LIN {X 0.064,Y -465.840,Z 820.018,A 0.000,B 0.000,C 90.000,E1 219.277} C_DIS
LIN {X -0.205,Y -462.583,Z 820.010,A 0.000,B 0.000,C 90.000,E1 217.729} C_DIS
LIN {X 0.196,Y -459.320,Z 820.001,A 0.000,B 0.000,C 90.000,E1 216.091} C_DIS
LIN {X -0.112,Y -456.022,Z 819.992,A 0.000,B 0.000,C 90.000,E1 214.532} C_DIS
LIN {X 0.155,Y -450.639,Z 819.978,A 0.000,B 0.000,C 90.000,E1 211.926} C_DIS
LIN {X 0.021,Y -446.616,Z 819.967,A 0.000,B 0.000,C 90.000,E1 210.001} C_DIS
LIN {X 0.126,Y -443.411,Z 819.958,A 0.000,B 0.000,C 90.000,E1 208.359} C_DIS
LIN {X -0.002,Y -439.571,Z 819.947,A 0.000,B 0.000,C 90.000,E1 206.411} C_DIS
LIN {X 0.099,Y -437.621,Z 819.941,A 0.000,B 0.000,C 90.000,E1 205.412} C_DIS
LIN {X 0.024,Y -434.306,Z 819.932,A 0.000,B 0.000,C 90.000,E1 203.770} C_DIS
LIN {X 0.087,Y -430.412,Z 819.921,A 0.000,B 0.000,C 90.000,E1 201.770} C_DIS
LIN {X 0.138,Y -426.596,Z 819.910,A 0.000,B 0.000,C 90.000,E1 199.758} C_DIS
LIN {X -0.092,Y -423.266,Z 819.901,A 0.000,B 0.000,C 90.000,E1 198.109} C_DIS
LIN {X -0.075,Y -419.349,Z 819.889,A 0.000,B 0.000,C 90.000,E1 196.079} C_DIS
LIN {X 0.146,Y -415.472,Z 819.878,A 0.000,B 0.000,C 90.000,E1 194.008} C_DIS
LIN {X 0.141,Y -412.294,Z 819.868,A 0.000,B 0.000,C 90.000,E1 192.299} C_DIS
LIN {X 0.007,Y -408.308,Z 819.857,A 0.000,B 0.000,C 90.000,E1 190.254} C_DIS
LIN {X 0.096,Y -405.067,Z 819.847,A 0.000,B 0.000,C 90.000,E1 188.511} C_DIS
LIN {X 0.058,Y -401.826,Z 819.838,A 0.000,B 0.000,C 90.000,E1 186.777} C_DIS
LIN {X 0.025,Y -395.279,Z 819.816,A 0.000,B 0.000,C 90.000,E1 182.922} C_DIS
LIN {X 0.015,Y -392.207,Z 819.805,A 0.000,B 0.000,C 90.000,E1 180.802} C_DIS
LIN {X 0.152,Y -388.677,Z 819.789,A 0.000,B 0.000,C 90.000,E1 177.936} C_DIS
LIN {X 0.084,Y -386.545,Z 819.779,A 0.000,B 0.000,C 90.000,E1 176.159} C_DIS
LIN {X -0.093,Y -384.076,Z 819.767,A 0.000,B 0.000,C 90.000,E1 174.033} C_DIS
LIN {X -0.125,Y -380.731,Z 819.749,A 0.000,B 0.000,C 90.000,E1 170.792} C_DIS
LIN {X 0.144,Y -378.740,Z 819.737,A 0.000,B 0.000,C 90.000,E1 168.578} C_DIS
LIN {X -0.067,Y -376.335,Z 819.721,A 0.000,B 0.000,C 90.000,E1 165.700} C_DIS
LIN {X 0.130,Y -373.483,Z 819.682,A 0.000,B 0.000,C 90.000,E1 158.720} C_DIS
LIN {X -0.016,Y -374.195,Z 819.668,A 0.000,B 0.000,C 90.000,E1 156.177} C_DIS
LIN {X 0.047,Y -376.178,Z 819.656,A 0.000,B 0.000,C 90.000,E1 153.973} C_DIS
LIN {X -0.036,Y -377.112,Z 819.651,A 0.000,B 0.000,C 90.000,E1 153.256} C_DIS
LIN {X 0.026,Y -379.071,Z 819.645,A 0.000,B 0.000,C 90.000,E1 152.153} C_DIS
LIN {X -0.028,Y -380.633,Z 819.641,A 0.000,B 0.000,C 90.000,E1 151.435} C_DIS
LIN {X 0.156,Y -383.722,Z 819.635,A 0.000,B 0.000,C 90.000,E1 150.333} C_DIS
LIN {X 0.046,Y -384.906,Z 819.633,A 0.000,B 0.000,C 90.000,E1 149.999} C_DIS
LIN {X 0.035,Y -387.998,Z 819.629,A 0.000,B 0.000,C 90.000,E1 149.282} C_DIS
LIN {X -0.197,Y -390.381,Z 819.627,A 0.000,B 0.000,C 90.000,E1 148.869} C_DIS
LIN {X 0.187,Y -392.330,Z 819.625,A 0.000,B 0.000,C 90.000,E1 148.456} C_DIS
LIN {X 0.040,Y -394.553,Z 819.623,A 0.000,B 0.000,C 90.000,E1 148.122} C_DIS
LIN {X -0.108,Y -399.019,Z 819.620,A 0.000,B 0.000,C 90.000,E1 147.582} C_DIS
LIN {X -0.132,Y -406.021,Z 819.616,A 0.000,B 0.000,C 90.000,E1 146.834} C_DIS
LIN {X 0.106,Y -413.015,Z 819.612,A 0.000,B 0.000,C 90.000,E1 146.215} C_DIS
LIN {X 0.082,Y -426.154,Z 819.607,A 0.000,B 0.000,C 90.000,E1 145.261} C_DIS
LIN {X -0.035,Y -435.967,Z 819.603,A 0.000,B 0.000,C 90.000,E1 144.609} C_DIS
LIN {X -0.214,Y -446.937,Z 819.599,A 0.000,B 0.000,C 90.000,E1 143.783} C_DIS
LIN {X 0.166,Y -452.778,Z 819.596,A 0.000,B 0.000,C 90.000,E1 143.210} C_DIS
LIN {X -0.262,Y -456.921,Z 819.593,A 0.000,B 0.000,C 90.000,E1 142.844} C_DIS
LIN {X 0.206,Y -462.297,Z 819.590,A 0.000,B 0.000,C 90.000,E1 142.190} C_DIS
LIN {X -0.274,Y -471.185,Z 819.584,A 0.000,B 0.000,C 90.000,E1 141.170} C_DIS
LIN {X 0.222,Y -474.561,Z 819.582,A 0.000,B 0.000,C 90.000,E1 140.642} C_DIS
LIN {X 0.087,Y -477.926,Z 819.579,A 0.000,B 0.000,C 90.000,E1 140.194} C_DIS
LIN {X -0.230,Y -483.509,Z 819.575,A 0.000,B 0.000,C 90.000,E1 139.461} C_DIS
LIN {X -0.288,Y -487.498,Z 819.571,A 0.000,B 0.000,C 90.000,E1 138.852} C_DIS
LIN {X -0.067,Y -490.481,Z 819.569,A 0.000,B 0.000,C 90.000,E1 138.366} C_DIS
LIN {X 0.018,Y -494.875,Z 819.564,A 0.000,B 0.000,C 90.000,E1 137.595} C_DIS
LIN {X 0.001,Y -500.954,Z 819.559,A 0.000,B 0.000,C 90.000,E1 136.539} C_DIS
LIN {X -0.074,Y -505.578,Z 819.554,A 0.000,B 0.000,C 90.000,E1 135.648} C_DIS
LIN {X 0.026,Y -508.795,Z 819.550,A 0.000,B 0.000,C 90.000,E1 135.040} C_DIS
LIN {X -0.194,Y -513.933,Z 819.545,A 0.000,B 0.000,C 90.000,E1 134.028} C_DIS
LIN {X -0.063,Y -520.525,Z 819.537,A 0.000,B 0.000,C 90.000,E1 132.690} C_DIS
LIN {X 0.164,Y -523.164,Z 819.534,A 0.000,B 0.000,C 90.000,E1 132.081} C_DIS
LIN {X 0.094,Y -528.588,Z 819.527,A 0.000,B 0.000,C 90.000,E1 130.782} C_DIS
LIN {X -0.065,Y -532.865,Z 819.520,A 0.000,B 0.000,C 90.000,E1 129.644} C_DIS
LIN {X 0.246,Y -536.671,Z 819.514,A 0.000,B 0.000,C 90.000,E1 128.463} C_DIS
LIN {X -0.158,Y -539.163,Z 819.509,A 0.000,B 0.000,C 90.000,E1 127.649} C_DIS
LIN {X -0.112,Y -541.425,Z 819.504,A 0.000,B 0.000,C 90.000,E1 126.790} C_DIS
LIN {X -0.066,Y -542.850,Z 819.501,A 0.000,B 0.000,C 90.000,E1 126.217} C_DIS
LIN {X -0.011,Y -544.045,Z 819.498,A 0.000,B 0.000,C 90.000,E1 125.644} C_DIS
LIN {X -0.263,Y -544.826,Z 819.495,A 0.000,B 0.000,C 90.000,E1 125.105} C_DIS
LIN {X -0.194,Y -545.485,Z 819.492,A 0.000,B 0.000,C 90.000,E1 124.532} C_DIS
LIN {X 0.133,Y -546.070,Z 819.484,A 0.000,B 0.000,C 90.000,E1 123.086} C_DIS
LIN {X -0.318,Y -547.175,Z 819.478,A 0.000,B 0.000,C 90.000,E1 122.005} C_DIS
LIN {X -0.036,Y -547.993,Z 819.473,A 0.000,B 0.000,C 90.000,E1 121.131} C_DIS
LIN {X -0.253,Y -548.782,Z 819.470,A 0.000,B 0.000,C 90.000,E1 120.590} C_DIS
LIN {X 0.253,Y -549.304,Z 819.468,A 0.000,B 0.000,C 90.000,E1 120.256} C_DIS
LIN {X 0.009,Y -549.680,Z 819.467,A 0.000,B 0.000,C 90.000,E1 120.001} C_DIS
LIN {X -0.078,Y -550.090,Z 819.464,A 0.000,B 0.000,C 90.000,E1 119.589} C_DIS
LIN {X 0.045,Y -550.848,Z 819.462,A 0.000,B 0.000,C 90.000,E1 119.155} C_DIS
LIN {X -0.044,Y -551.594,Z 819.461,A 0.000,B 0.000,C 90.000,E1 119.027} C_DIS
LIN {X -0.011,Y -552.319,Z 819.460,A 0.000,B 0.000,C 90.000,E1 118.743} C_DIS
LIN {X -0.094,Y -552.319,Z 819.458,A 0.000,B 0.000,C 90.000,E1 118.437} C_DIS
LIN {X 0.001,Y -552.285,Z 819.458,A 0.000,B 0.000,C 90.000,E1 118.409} C_DIS
LIN {X -0.042,Y -552.280,Z 819.458,A 0.000,B 0.000,C 90.000,E1 118.409} C_DIS
LIN {X 0.017,Y -552.707,Z 819.457,A 0.000,B 0.000,C 90.000,E1 118.180} C_DIS
LIN {X 0.050,Y -553.492,Z 819.455,A 0.000,B 0.000,C 90.000,E1 117.897} C_DIS
LIN {X -0.064,Y -553.553,Z 819.454,A 0.000,B 0.000,C 90.000,E1 117.769} C_DIS
LIN {X -0.131,Y -554.947,Z 819.450,A 0.000,B 0.000,C 90.000,E1 117.078} C_DIS
LIN {X -0.256,Y -556.790,Z 819.444,A 0.000,B 0.000,C 90.000,E1 115.976} C_DIS
LIN {X 0.136,Y -558.183,Z 819.438,A 0.000,B 0.000,C 90.000,E1 114.823} C_DIS
LIN {X -0.121,Y -559.816,Z 819.430,A 0.000,B 0.000,C 90.000,E1 113.462} C_DIS
LIN {X -0.127,Y -561.223,Z 819.423,A 0.000,B 0.000,C 90.000,E1 112.078} C_DIS
LIN {X -0.124,Y -562.087,Z 819.417,A 0.000,B 0.000,C 90.000,E1 110.972} C_DIS
LIN {X -0.112,Y -562.630,Z 819.410,A 0.000,B 0.000,C 90.000,E1 109.866} C_DIS
LIN {X -0.147,Y -562.902,Z 819.403,A 0.000,B 0.000,C 90.000,E1 108.489} C_DIS
LIN {X 0.070,Y -563.250,Z 819.390,A 0.000,B 0.000,C 90.000,E1 106.260} C_DIS
LIN {X 0.206,Y -564.671,Z 819.372,A 0.000,B 0.000,C 90.000,E1 102.939} C_DIS
LIN {X 0.268,Y -565.893,Z 819.361,A 0.000,B 0.000,C 90.000,E1 101.007} C_DIS
LIN {X 0.159,Y -567.308,Z 819.351,A 0.000,B 0.000,C 90.000,E1 99.095} C_DIS
LIN {X -0.005,Y -568.419,Z 819.342,A 0.000,B 0.000,C 90.000,E1 97.466} C_DIS
LIN {X 0.262,Y -569.428,Z 819.332,A 0.000,B 0.000,C 90.000,E1 95.796} C_DIS
LIN {X -0.063,Y -570.191,Z 819.323,A 0.000,B 0.000,C 90.000,E1 94.188} C_DIS
LIN {X 0.069,Y -570.727,Z 819.316,A 0.000,B 0.000,C 90.000,E1 92.808} C_DIS
LIN {X 0.043,Y -571.139,Z 819.310,A 0.000,B 0.000,C 90.000,E1 91.718} C_DIS
LIN {X 0.141,Y -571.612,Z 819.302,A 0.000,B 0.000,C 90.000,E1 90.344} C_DIS
LIN {X -0.048,Y -572.109,Z 819.291,A 0.000,B 0.000,C 90.000,E1 88.453} C_DIS
LIN {X 0.081,Y -572.499,Z 819.284,A 0.000,B 0.000,C 90.000,E1 87.078} C_DIS
LIN {X -0.009,Y -572.878,Z 819.273,A 0.000,B 0.000,C 90.000,E1 85.179} C_DIS
LIN {X -0.082,Y -573.162,Z 819.263,A 0.000,B 0.000,C 90.000,E1 83.280} C_DIS
LIN {X -0.206,Y -573.573,Z 819.254,A 0.000,B 0.000,C 90.000,E1 81.659} C_DIS
LIN {X 0.242,Y -574.013,Z 819.245,A 0.000,B 0.000,C 90.000,E1 79.982} C_DIS
LIN {X 0.331,Y -574.389,Z 819.235,A 0.000,B 0.000,C 90.000,E1 78.342} C_DIS
LIN {X 0.231,Y -574.657,Z 819.228,A 0.000,B 0.000,C 90.000,E1 76.992} C_DIS
LIN {X -0.229,Y -574.764,Z 819.219,A 0.000,B 0.000,C 90.000,E1 75.408} C_DIS
LIN {X -0.043,Y -574.803,Z 819.211,A 0.000,B 0.000,C 90.000,E1 74.031} C_DIS
LIN {X -0.018,Y -574.673,Z 819.201,A 0.000,B 0.000,C 90.000,E1 72.127} C_DIS
LIN {X -0.198,Y -574.365,Z 819.190,A 0.000,B 0.000,C 90.000,E1 70.242} C_DIS
LIN {X -0.011,Y -573.965,Z 819.181,A 0.000,B 0.000,C 90.000,E1 68.592} C_DIS
LIN {X 0.008,Y -573.527,Z 819.174,A 0.000,B 0.000,C 90.000,E1 67.230} C_DIS
LIN {X 0.013,Y -572.980,Z 819.166,A 0.000,B 0.000,C 90.000,E1 65.869} C_DIS
LIN {X -0.282,Y -572.384,Z 819.158,A 0.000,B 0.000,C 90.000,E1 64.537} C_DIS
LIN {X 0.180,Y -571.631,Z 819.151,A 0.000,B 0.000,C 90.000,E1 63.127} C_DIS
LIN {X 0.288,Y -570.867,Z 819.145,A 0.000,B 0.000,C 90.000,E1 62.025} C_DIS
LIN {X -0.114,Y -569.952,Z 819.139,A 0.000,B 0.000,C 90.000,E1 60.973} C_DIS
LIN {X -0.033,Y -568.780,Z 819.133,A 0.000,B 0.000,C 90.000,E1 59.871} C_DIS
LIN {X -0.178,Y -567.446,Z 819.127,A 0.000,B 0.000,C 90.000,E1 58.791} C_DIS
LIN {X 0.251,Y -565.487,Z 819.119,A 0.000,B 0.000,C 90.000,E1 57.375} C_DIS
LIN {X 0.060,Y -563.654,Z 819.113,A 0.000,B 0.000,C 90.000,E1 56.294} C_DIS
LIN {X 0.153,Y -561.489,Z 819.107,A 0.000,B 0.000,C 90.000,E1 55.182} C_DIS
LIN {X -0.242,Y -559.066,Z 819.101,A 0.000,B 0.000,C 90.000,E1 54.116} C_DIS
LIN {X 0.030,Y -557.004,Z 819.096,A 0.000,B 0.000,C 90.000,E1 53.256} C_DIS
LIN {X -0.061,Y -554.683,Z 819.091,A 0.000,B 0.000,C 90.000,E1 52.431} C_DIS
LIN {X -0.282,Y -552.076,Z 819.087,A 0.000,B 0.000,C 90.000,E1 51.618} C_DIS
LIN {X 0.191,Y -550.176,Z 819.084,A 0.000,B 0.000,C 90.000,E1 51.009} C_DIS
LIN {X -0.069,Y -546.997,Z 819.079,A 0.000,B 0.000,C 90.000,E1 50.194} C_DIS
LIN {X 0.050,Y -543.508,Z 819.074,A 0.000,B 0.000,C 90.000,E1 49.337} C_DIS
LIN {X 0.047,Y -540.939,Z 819.071,A 0.000,B 0.000,C 90.000,E1 48.771} C_DIS
LIN {X -0.328,Y -538.176,Z 819.068,A 0.000,B 0.000,C 90.000,E1 48.243} C_DIS
LIN {X 0.211,Y -534.326,Z 819.064,A 0.000,B 0.000,C 90.000,E1 47.472} C_DIS
LIN {X 0.151,Y -530.947,Z 819.061,A 0.000,B 0.000,C 90.000,E1 46.905} C_DIS
LIN {X -0.294,Y -527.208,Z 819.057,A 0.000,B 0.000,C 90.000,E1 46.377} C_DIS
LIN {X -0.025,Y -523.059,Z 819.054,A 0.000,B 0.000,C 90.000,E1 45.769} C_DIS
LIN {X 0.066,Y -518.885,Z 819.051,A 0.000,B 0.000,C 90.000,E1 45.202} C_DIS
LIN {X 0.048,Y -514.196,Z 819.048,A 0.000,B 0.000,C 90.000,E1 44.636} C_DIS
LIN {X -0.274,Y -507.621,Z 819.044,A 0.000,B 0.000,C 90.000,E1 43.947} C_DIS
LIN {X 0.209,Y -503.531,Z 819.042,A 0.000,B 0.000,C 90.000,E1 43.461} C_DIS
LIN {X 0.086,Y -499.288,Z 819.039,A 0.000,B 0.000,C 90.000,E1 43.056} C_DIS
LIN {X -0.048,Y -492.095,Z 819.036,A 0.000,B 0.000,C 90.000,E1 42.405} C_DIS
LIN {X 0.065,Y -484.633,Z 819.032,A 0.000,B 0.000,C 90.000,E1 41.757} C_DIS
LIN {X 0.006,Y -478.368,Z 819.029,A 0.000,B 0.000,C 90.000,E1 41.272} C_DIS
LIN {X -0.144,Y -470.550,Z 819.026,A 0.000,B 0.000,C 90.000,E1 40.701} C_DIS
LIN {X 0.100,Y -453.134,Z 819.019,A 0.000,B 0.000,C 90.000,E1 39.402} C_DIS
LIN {X -0.118,Y -424.777,Z 819.007,A 0.000,B 0.000,C 90.000,E1 37.317} C_DIS
LIN {X -0.016,Y -409.437,Z 819.000,A 0.000,B 0.000,C 90.000,E1 36.011} C_DIS
LIN {X 0.126,Y -402.370,Z 818.996,A 0.000,B 0.000,C 90.000,E1 35.311} C_DIS
LIN {X -0.153,Y -398.570,Z 818.994,A 0.000,B 0.000,C 90.000,E1 34.898} C_DIS
LIN {X -0.191,Y -398.539,Z 818.994,A 0.000,B 0.000,C 90.000,E1 34.898} C_DIS
LIN {X 0.065,Y -394.044,Z 818.978,A 0.000,B 0.000,C 90.000,E1 32.005} C_DIS
LIN {X 0.063,Y -392.608,Z 818.974,A 0.000,B 0.000,C 90.000,E1 31.209} C_DIS
LIN {X -0.108,Y -393.788,Z 818.958,A 0.000,B 0.000,C 90.000,E1 28.487} C_DIS
LIN {X -0.013,Y -395.477,Z 818.943,A 0.000,B 0.000,C 90.000,E1 25.643} C_DIS
LIN {X 0.126,Y -397.180,Z 818.929,A 0.000,B 0.000,C 90.000,E1 23.153} C_DIS
LIN {X 0.101,Y -399.800,Z 818.911,A 0.000,B 0.000,C 90.000,E1 19.993} C_DIS
LIN {X 0.170,Y -404.433,Z 818.888,A 0.000,B 0.000,C 90.000,E1 15.788} C_DIS
LIN {X -0.101,Y -408.925,Z 818.871,A 0.000,B 0.000,C 90.000,E1 12.703} C_DIS
LIN {X 0.127,Y -412.414,Z 818.859,A 0.000,B 0.000,C 90.000,E1 10.602} C_DIS
LIN {X 0.011,Y -416.583,Z 818.846,A 0.000,B 0.000,C 90.000,E1 8.219} C_DIS
LIN {X -0.172,Y -420.297,Z 818.834,A 0.000,B 0.000,C 90.000,E1 6.201} C_DIS
LIN {X 0.118,Y -424.066,Z 818.823,A 0.000,B 0.000,C 90.000,E1 4.131} C_DIS
LIN {X 0.126,Y -428.656,Z 818.810,A 0.000,B 0.000,C 90.000,E1 1.776} C_DIS
LIN {X -0.098,Y -434.381,Z 818.795,A 0.000,B 0.000,C 90.000,E1 359.141} C_DIS
LIN {X -0.147,Y -440.536,Z 818.781,A 0.000,B 0.000,C 90.000,E1 356.502} C_DIS
LIN {X 0.215,Y -445.329,Z 818.770,A 0.000,B 0.000,C 90.000,E1 354.489} C_DIS
LIN {X -0.205,Y -450.296,Z 818.759,A 0.000,B 0.000,C 90.000,E1 352.591} C_DIS
LIN {X 0.142,Y -453.740,Z 818.752,A 0.000,B 0.000,C 90.000,E1 351.254} C_DIS
LIN {X 0.189,Y -456.426,Z 818.747,A 0.000,B 0.000,C 90.000,E1 350.443} C_DIS
LIN {X -0.041,Y -457.795,Z 818.745,A 0.000,B 0.000,C 90.000,E1 350.151} C_DIS
LIN {X 0.188,Y -459.714,Z 818.744,A 0.000,B 0.000,C 90.000,E1 349.803} C_DIS
LIN {X -0.030,Y -462.146,Z 818.742,A 0.000,B 0.000,C 90.000,E1 349.511} C_DIS
LIN {X 0.047,Y -463.622,Z 818.741,A 0.000,B 0.000,C 90.000,E1 349.342} C_DIS
LIN {X 0.000,Y -468.296,Z 818.739,A 0.000,B 0.000,C 90.000,E1 348.926} C_DIS
LIN {X 0.276,Y -475.809,Z 818.735,A 0.000,B 0.000,C 90.000,E1 348.342} C_DIS
LIN {X 0.107,Y -491.394,Z 818.730,A 0.000,B 0.000,C 90.000,E1 347.353} C_DIS
LIN {X -0.258,Y -499.351,Z 818.727,A 0.000,B 0.000,C 90.000,E1 346.881} C_DIS
LIN {X 0.108,Y -512.060,Z 818.722,A 0.000,B 0.000,C 90.000,E1 345.992} C_DIS
LIN {X -0.288,Y -524.419,Z 818.717,A 0.000,B 0.000,C 90.000,E1 345.172} C_DIS
LIN {X -0.113,Y -535.161,Z 818.713,A 0.000,B 0.000,C 90.000,E1 344.393} C_DIS
LIN {X 0.163,Y -543.988,Z 818.710,A 0.000,B 0.000,C 90.000,E1 343.685} C_DIS
LIN {X -0.186,Y -549.737,Z 818.707,A 0.000,B 0.000,C 90.000,E1 343.251} C_DIS
LIN {X 0.308,Y -556.798,Z 818.704,A 0.000,B 0.000,C 90.000,E1 342.598} C_DIS
LIN {X 0.235,Y -559.566,Z 818.702,A 0.000,B 0.000,C 90.000,E1 342.362} C_DIS
LIN {X -0.109,Y -566.064,Z 818.699,A 0.000,B 0.000,C 90.000,E1 341.764} C_DIS
LIN {X 0.105,Y -571.119,Z 818.696,A 0.000,B 0.000,C 90.000,E1 341.221} C_DIS
LIN {X 0.202,Y -577.132,Z 818.692,A 0.000,B 0.000,C 90.000,E1 340.550} C_DIS
LIN {X -0.245,Y -580.537,Z 818.690,A 0.000,B 0.000,C 90.000,E1 340.188} C_DIS
LIN {X -0.005,Y -584.747,Z 818.687,A 0.000,B 0.000,C 90.000,E1 339.625} C_DIS
LIN {X 0.000,Y -589.612,Z 818.683,A 0.000,B 0.000,C 90.000,E1 338.954} C_DIS
LIN {X 0.101,Y -593.242,Z 818.680,A 0.000,B 0.000,C 90.000,E1 338.411} C_DIS
LIN {X 0.127,Y -598.251,Z 818.676,A 0.000,B 0.000,C 90.000,E1 337.614} C_DIS
LIN {X 0.127,Y -604.634,Z 818.670,A 0.000,B 0.000,C 90.000,E1 336.561} C_DIS
LIN {X -0.115,Y -611.479,Z 818.663,A 0.000,B 0.000,C 90.000,E1 335.409} C_DIS
LIN {X 0.068,Y -616.650,Z 818.658,A 0.000,B 0.000,C 90.000,E1 334.485} C_DIS
LIN {X 0.013,Y -622.075,Z 818.653,A 0.000,B 0.000,C 90.000,E1 333.461} C_DIS
LIN {X 0.025,Y -626.619,Z 818.648,A 0.000,B 0.000,C 90.000,E1 332.564} C_DIS
LIN {X -0.174,Y -630.858,Z 818.643,A 0.000,B 0.000,C 90.000,E1 331.691} C_DIS
LIN {X -0.083,Y -634.400,Z 818.638,A 0.000,B 0.000,C 90.000,E1 330.923} C_DIS
LIN {X -0.108,Y -640.068,Z 818.631,A 0.000,B 0.000,C 90.000,E1 329.665} C_DIS
LIN {X -0.165,Y -643.186,Z 818.627,A 0.000,B 0.000,C 90.000,E1 328.918} C_DIS
LIN {X -0.118,Y -647.110,Z 818.622,A 0.000,B 0.000,C 90.000,E1 327.916} C_DIS
LIN {X -0.102,Y -649.896,Z 818.618,A 0.000,B 0.000,C 90.000,E1 327.168} C_DIS
LIN {X 0.021,Y -653.278,Z 818.612,A 0.000,B 0.000,C 90.000,E1 326.167} C_DIS
LIN {X 0.005,Y -656.498,Z 818.607,A 0.000,B 0.000,C 90.000,E1 325.182} C_DIS
LIN {X -0.412,Y -660.115,Z 818.600,A 0.000,B 0.000,C 90.000,E1 323.989} C_DIS
LIN {X 0.061,Y -662.884,Z 818.594,A 0.000,B 0.000,C 90.000,E1 322.970} C_DIS
LIN {X -0.326,Y -664.721,Z 818.590,A 0.000,B 0.000,C 90.000,E1 322.271} C_DIS
LIN {X 0.210,Y -666.998,Z 818.585,A 0.000,B 0.000,C 90.000,E1 321.251} C_DIS
LIN {X 0.261,Y -669.150,Z 818.579,A 0.000,B 0.000,C 90.000,E1 320.275} C_DIS
LIN {X 0.343,Y -671.150,Z 818.574,A 0.000,B 0.000,C 90.000,E1 319.299} C_DIS
LIN {X 0.015,Y -673.470,Z 818.567,A 0.000,B 0.000,C 90.000,E1 318.119} C_DIS
LIN {X 0.072,Y -674.802,Z 818.563,A 0.000,B 0.000,C 90.000,E1 317.391} C_DIS
LIN {X -0.254,Y -676.645,Z 818.557,A 0.000,B 0.000,C 90.000,E1 316.215} C_DIS
LIN {X -0.154,Y -677.717,Z 818.553,A 0.000,B 0.000,C 90.000,E1 315.486} C_DIS
LIN {X -0.041,Y -678.688,Z 818.549,A 0.000,B 0.000,C 90.000,E1 314.757} C_DIS
LIN {X 0.164,Y -680.193,Z 818.542,A 0.000,B 0.000,C 90.000,E1 313.542} C_DIS
LIN {X -0.036,Y -681.891,Z 818.534,A 0.000,B 0.000,C 90.000,E1 312.123} C_DIS
LIN {X -0.150,Y -683.438,Z 818.526,A 0.000,B 0.000,C 90.000,E1 310.701} C_DIS
LIN {X -0.226,Y -684.931,Z 818.518,A 0.000,B 0.000,C 90.000,E1 309.277} C_DIS
LIN {X 0.254,Y -686.296,Z 818.510,A 0.000,B 0.000,C 90.000,E1 307.810} C_DIS
LIN {X -0.030,Y -687.700,Z 818.501,A 0.000,B 0.000,C 90.000,E1 306.171} C_DIS
LIN {X 0.078,Y -688.817,Z 818.493,A 0.000,B 0.000,C 90.000,E1 304.739} C_DIS
LIN {X 0.371,Y -689.821,Z 818.485,A 0.000,B 0.000,C 90.000,E1 303.293} C_DIS
LIN {X -0.046,Y -691.000,Z 818.476,A 0.000,B 0.000,C 90.000,E1 301.671} C_DIS
LIN {X 0.047,Y -691.765,Z 818.471,A 0.000,B 0.000,C 90.000,E1 300.718} C_DIS
LIN {X -0.091,Y -692.888,Z 818.462,A 0.000,B 0.000,C 90.000,E1 299.077} C_DIS
LIN {X 0.161,Y -693.875,Z 818.454,A 0.000,B 0.000,C 90.000,E1 297.641} C_DIS
LIN {X 0.364,Y -695.143,Z 818.445,A 0.000,B 0.000,C 90.000,E1 295.976} C_DIS
LIN {X 0.042,Y -696.279,Z 818.437,A 0.000,B 0.000,C 90.000,E1 294.591} C_DIS
LIN {X 0.298,Y -696.456,Z 818.435,A 0.000,B 0.000,C 90.000,E1 294.335} C_DIS
LIN {X 0.146,Y -696.298,Z 818.431,A 0.000,B 0.000,C 90.000,E1 293.643} C_DIS
LIN {X -0.262,Y -695.128,Z 818.429,A 0.000,B 0.000,C 90.000,E1 293.206} C_DIS
LIN {X -0.011,Y -694.378,Z 818.428,A 0.000,B 0.000,C 90.000,E1 292.950} C_DIS
LIN {X 0.112,Y -693.656,Z 818.427,A 0.000,B 0.000,C 90.000,E1 292.823} C_DIS
LIN {X -0.033,Y -692.660,Z 818.426,A 0.000,B 0.000,C 90.000,E1 292.717} C_DIS
LIN {X 0.352,Y -689.102,Z 818.424,A 0.000,B 0.000,C 90.000,E1 292.333} C_DIS
LIN {X -0.142,Y -687.796,Z 818.424,A 0.000,B 0.000,C 90.000,E1 292.259} C_DIS
LIN {X -0.211,Y -685.865,Z 818.423,A 0.000,B 0.000,C 90.000,E1 292.153} C_DIS
LIN {X -0.006,Y -681.676,Z 818.422,A 0.000,B 0.000,C 90.000,E1 291.950} C_DIS
LIN {X -0.377,Y -678.102,Z 818.421,A 0.000,B 0.000,C 90.000,E1 291.844} C_DIS
LIN {X -0.218,Y -672.525,Z 818.420,A 0.000,B 0.000,C 90.000,E1 291.663} C_DIS
LIN {X 0.219,Y -663.517,Z 818.419,A 0.000,B 0.000,C 90.000,E1 291.461} C_DIS
LIN {X 0.186,Y -645.614,Z 818.418,A 0.000,B 0.000,C 90.000,E1 291.173} C_DIS
LIN {X 0.227,Y -635.221,Z 818.417,A 0.000,B 0.000,C 90.000,E1 290.972} C_DIS
LIN {X -0.180,Y -625.486,Z 818.415,A 0.000,B 0.000,C 90.000,E1 290.791} C_DIS
LIN {X 0.041,Y -619.557,Z 818.415,A 0.000,B 0.000,C 90.000,E1 290.610} C_DIS
LIN {X 0.065,Y -612.527,Z 818.413,A 0.000,B 0.000,C 90.000,E1 290.355} C_DIS
LIN {X 0.090,Y -609.015,Z 818.412,A 0.000,B 0.000,C 90.000,E1 290.194} C_DIS
LIN {X 0.055,Y -605.447,Z 818.411,A 0.000,B 0.000,C 90.000,E1 289.993} C_DIS
LIN {X 0.000,Y -605.415,Z 818.411,A 0.000,B 0.000,C 90.000,E1 289.993} C_DIS
LIN {X -0.001,Y -604.757,Z 818.411,A 0.000,B 0.000,C 90.000,E1 289.885} C_DIS
LIN {X -0.210,Y -603.719,Z 818.410,A 0.000,B 0.000,C 90.000,E1 289.758} C_DIS
LIN {X -0.115,Y -603.883,Z 818.408,A 0.000,B 0.000,C 90.000,E1 289.504} C_DIS
LIN {X -0.357,Y -604.282,Z 818.408,A 0.000,B 0.000,C 90.000,E1 289.396} C_DIS
LIN {X -0.254,Y -606.323,Z 818.405,A 0.000,B 0.000,C 90.000,E1 288.960} C_DIS
LIN {X 0.009,Y -608.787,Z 818.403,A 0.000,B 0.000,C 90.000,E1 288.544} C_DIS
LIN {X 0.254,Y -612.122,Z 818.400,A 0.000,B 0.000,C 90.000,E1 288.000} C_DIS
LIN {X -0.279,Y -615.641,Z 818.397,A 0.000,B 0.000,C 90.000,E1 287.402} C_DIS
LIN {X -0.224,Y -619.003,Z 818.392,A 0.000,B 0.000,C 90.000,E1 286.622} C_DIS
LIN {X -0.138,Y -621.783,Z 818.388,A 0.000,B 0.000,C 90.000,E1 285.843} C_DIS
LIN {X 0.024,Y -623.265,Z 818.385,A 0.000,B 0.000,C 90.000,E1 285.315} C_DIS
LIN {X 0.151,Y -625.114,Z 818.381,A 0.000,B 0.000,C 90.000,E1 284.537} C_DIS
LIN {X -0.264,Y -625.907,Z 818.378,A 0.000,B 0.000,C 90.000,E1 284.064} C_DIS
LIN {X -0.066,Y -626.486,Z 818.375,A 0.000,B 0.000,C 90.000,E1 283.536} C_DIS
LIN {X -0.063,Y -626.946,Z 818.371,A 0.000,B 0.000,C 90.000,E1 282.771} C_DIS
LIN {X 0.146,Y -626.576,Z 818.368,A 0.000,B 0.000,C 90.000,E1 282.243} C_DIS
LIN {X 0.148,Y -625.448,Z 818.364,A 0.000,B 0.000,C 90.000,E1 281.478} C_DIS
LIN {X -0.269,Y -624.308,Z 818.361,A 0.000,B 0.000,C 90.000,E1 281.007} C_DIS
LIN {X -0.197,Y -622.920,Z 818.358,A 0.000,B 0.000,C 90.000,E1 280.489} C_DIS
LIN {X -0.019,Y -621.143,Z 818.355,A 0.000,B 0.000,C 90.000,E1 279.962} C_DIS
LIN {X -0.024,Y -618.293,Z 818.352,A 0.000,B 0.000,C 90.000,E1 279.321} C_DIS
LIN {X 0.016,Y -615.359,Z 818.349,A 0.000,B 0.000,C 90.000,E1 278.803} C_DIS
LIN {X 0.127,Y -611.931,Z 818.346,A 0.000,B 0.000,C 90.000,E1 278.276} C_DIS
LIN {X -0.216,Y -609.918,Z 818.345,A 0.000,B 0.000,C 90.000,E1 278.049} C_DIS
LIN {X -0.050,Y -606.491,Z 818.342,A 0.000,B 0.000,C 90.000,E1 277.644} C_DIS
LIN {X 0.162,Y -602.542,Z 818.340,A 0.000,B 0.000,C 90.000,E1 277.239} C_DIS
LIN {X 0.050,Y -601.135,Z 818.340,A 0.000,B 0.000,C 90.000,E1 277.125} C_DIS
LIN {X -0.291,Y -594.573,Z 818.337,A 0.000,B 0.000,C 90.000,E1 276.720} C_DIS
LIN {X 0.085,Y -591.033,Z 818.336,A 0.000,B 0.000,C 90.000,E1 276.486} C_DIS
LIN {X -0.151,Y -585.650,Z 818.335,A 0.000,B 0.000,C 90.000,E1 276.258} C_DIS
LIN {X -0.143,Y -580.431,Z 818.333,A 0.000,B 0.000,C 90.000,E1 276.030} C_DIS
LIN {X 0.186,Y -574.584,Z 818.332,A 0.000,B 0.000,C 90.000,E1 275.796} C_DIS
LIN {X -0.149,Y -568.345,Z 818.332,A 0.000,B 0.000,C 90.000,E1 275.682} C_DIS
LIN {X 0.115,Y -566.392,Z 818.331,A 0.000,B 0.000,C 90.000,E1 275.625} C_DIS
LIN {X -0.048,Y -561.313,Z 818.331,A 0.000,B 0.000,C 90.000,E1 275.625} C_DIS
LIN {X -0.080,Y -553.687,Z 818.331,A 0.000,B 0.000,C 90.000,E1 275.625} C_DIS
LIN {X 0.247,Y -551.917,Z 818.331,A 0.000,B 0.000,C 90.000,E1 275.568} C_DIS
LIN {X 0.215,Y -551.792,Z 818.331,A 0.000,B 0.000,C 90.000,E1 275.568} C_DIS
LIN {X 0.063,Y -550.067,Z 818.329,A 0.000,B 0.000,C 90.000,E1 275.277} C_DIS
LIN {X 0.013,Y -550.055,Z 818.329,A 0.000,B 0.000,C 90.000,E1 275.277} C_DIS
LIN {X -0.257,Y -547.943,Z 818.314,A 0.000,B 0.000,C 90.000,E1 272.465} C_DIS
LIN {X 0.083,Y -546.574,Z 818.303,A 0.000,B 0.000,C 90.000,E1 270.458} C_DIS
LIN {X -0.173,Y -545.183,Z 818.292,A 0.000,B 0.000,C 90.000,E1 268.511} C_DIS
LIN {X 0.142,Y -543.651,Z 818.279,A 0.000,B 0.000,C 90.000,E1 266.216} C_DIS
LIN {X -0.197,Y -542.798,Z 818.271,A 0.000,B 0.000,C 90.000,E1 264.837} C_DIS
LIN {X -0.038,Y -542.261,Z 818.267,A 0.000,B 0.000,C 90.000,E1 263.970} C_DIS
LIN {X 0.200,Y -540.797,Z 818.257,A 0.000,B 0.000,C 90.000,E1 262.243} C_DIS
LIN {X 0.017,Y -539.306,Z 818.248,A 0.000,B 0.000,C 90.000,E1 260.557} C_DIS
LIN {X 0.268,Y -537.902,Z 818.240,A 0.000,B 0.000,C 90.000,E1 259.106} C_DIS
LIN {X 0.122,Y -536.177,Z 818.230,A 0.000,B 0.000,C 90.000,E1 257.409} C_DIS
LIN {X 0.005,Y -534.713,Z 818.222,A 0.000,B 0.000,C 90.000,E1 255.992} C_DIS
LIN {X -0.138,Y -533.063,Z 818.214,A 0.000,B 0.000,C 90.000,E1 254.574} C_DIS
LIN {X 0.014,Y -531.097,Z 818.205,A 0.000,B 0.000,C 90.000,E1 252.834} C_DIS
LIN {X -0.060,Y -529.319,Z 818.197,A 0.000,B 0.000,C 90.000,E1 251.402} C_DIS
LIN {X -0.010,Y -527.896,Z 818.190,A 0.000,B 0.000,C 90.000,E1 250.242} C_DIS
LIN {X 0.196,Y -525.902,Z 818.182,A 0.000,B 0.000,C 90.000,E1 248.773} C_DIS
LIN {X 0.037,Y -523.373,Z 818.173,A 0.000,B 0.000,C 90.000,E1 247.050} C_DIS
LIN {X 0.016,Y -520.710,Z 818.163,A 0.000,B 0.000,C 90.000,E1 245.305} C_DIS
LIN {X -0.128,Y -518.814,Z 818.156,A 0.000,B 0.000,C 90.000,E1 244.152} C_DIS
LIN {X 0.068,Y -516.361,Z 818.148,A 0.000,B 0.000,C 90.000,E1 242.666} C_DIS
LIN {X -0.149,Y -515.391,Z 818.145,A 0.000,B 0.000,C 90.000,E1 242.103} C_DIS
LIN {X -0.127,Y -512.052,Z 818.135,A 0.000,B 0.000,C 90.000,E1 240.333} C_DIS
LIN {X -0.256,Y -509.343,Z 818.127,A 0.000,B 0.000,C 90.000,E1 238.869} C_DIS
LIN {X -0.064,Y -506.958,Z 818.120,A 0.000,B 0.000,C 90.000,E1 237.661} C_DIS
LIN {X 0.048,Y -505.134,Z 818.115,A 0.000,B 0.000,C 90.000,E1 236.755} C_DIS
LIN {X 0.049,Y -501.867,Z 818.107,A 0.000,B 0.000,C 90.000,E1 235.261} C_DIS
LIN {X -0.019,Y -499.109,Z 818.100,A 0.000,B 0.000,C 90.000,E1 234.069} C_DIS
LIN {X 0.297,Y -496.980,Z 818.095,A 0.000,B 0.000,C 90.000,E1 233.130} C_DIS
LIN {X -0.079,Y -493.298,Z 818.087,A 0.000,B 0.000,C 90.000,E1 231.662} C_DIS
LIN {X -0.017,Y -486.156,Z 818.070,A 0.000,B 0.000,C 90.000,E1 228.609} C_DIS
LIN {X -0.018,Y -481.253,Z 818.058,A 0.000,B 0.000,C 90.000,E1 226.458} C_DIS
LIN {X 0.029,Y -479.169,Z 818.053,A 0.000,B 0.000,C 90.000,E1 225.526} C_DIS
LIN {X 0.273,Y -475.783,Z 818.044,A 0.000,B 0.000,C 90.000,E1 223.947} C_DIS
LIN {X -0.212,Y -472.486,Z 818.036,A 0.000,B 0.000,C 90.000,E1 222.447} C_DIS
LIN {X -0.213,Y -467.882,Z 818.024,A 0.000,B 0.000,C 90.000,E1 220.253} C_DIS
LIN {X 0.018,Y -463.271,Z 818.011,A 0.000,B 0.000,C 90.000,E1 218.016} C_DIS
LIN {X 0.173,Y -459.362,Z 818.001,A 0.000,B 0.000,C 90.000,E1 216.091} C_DIS
LIN {X 0.028,Y -457.272,Z 817.995,A 0.000,B 0.000,C 90.000,E1 215.152} C_DIS
LIN {X -0.134,Y -456.062,Z 817.992,A 0.000,B 0.000,C 90.000,E1 214.532} C_DIS
LIN {X 0.045,Y -451.357,Z 817.979,A 0.000,B 0.000,C 90.000,E1 212.260} C_DIS
LIN {X -0.073,Y -447.326,Z 817.969,A 0.000,B 0.000,C 90.000,E1 210.335} C_DIS
LIN {X 0.050,Y -444.088,Z 817.959,A 0.000,B 0.000,C 90.000,E1 208.693} C_DIS
LIN {X -0.100,Y -440.908,Z 817.950,A 0.000,B 0.000,C 90.000,E1 207.078} C_DIS
LIN {X 0.245,Y -438.355,Z 817.943,A 0.000,B 0.000,C 90.000,E1 205.720} C_DIS
LIN {X 0.179,Y -435.064,Z 817.934,A 0.000,B 0.000,C 90.000,E1 204.079} C_DIS
LIN {X 0.096,Y -431.142,Z 817.923,A 0.000,B 0.000,C 90.000,E1 202.099} C_DIS
LIN {X -0.077,Y -427.317,Z 817.912,A 0.000,B 0.000,C 90.000,E1 200.120} C_DIS
LIN {X -0.081,Y -424.709,Z 817.904,A 0.000,B 0.000,C 90.000,E1 198.779} C_DIS
LIN {X 0.150,Y -420.119,Z 817.891,A 0.000,B 0.000,C 90.000,E1 196.386} C_DIS
LIN {X 0.095,Y -416.186,Z 817.880,A 0.000,B 0.000,C 90.000,E1 194.356} C_DIS
LIN {X 0.139,Y -412.398,Z 817.868,A 0.000,B 0.000,C 90.000,E1 192.299} C_DIS
LIN {X 0.007,Y -408.431,Z 817.857,A 0.000,B 0.000,C 90.000,E1 190.254} C_DIS
LIN {X 0.098,Y -405.198,Z 817.847,A 0.000,B 0.000,C 90.000,E1 188.511} C_DIS
LIN {X 0.063,Y -401.933,Z 817.838,A 0.000,B 0.000,C 90.000,E1 186.777} C_DIS
LIN {X 0.201,Y -397.043,Z 817.822,A 0.000,B 0.000,C 90.000,E1 183.955} C_DIS
LIN {X 0.102,Y -392.890,Z 817.807,A 0.000,B 0.000,C 90.000,E1 181.146} C_DIS
LIN {X 0.172,Y -388.846,Z 817.789,A 0.000,B 0.000,C 90.000,E1 177.936} C_DIS
LIN {X -0.179,Y -387.203,Z 817.781,A 0.000,B 0.000,C 90.000,E1 176.560} C_DIS
LIN {X -0.065,Y -384.310,Z 817.767,A 0.000,B 0.000,C 90.000,E1 174.033} C_DIS
LIN {X -0.174,Y -380.664,Z 817.747,A 0.000,B 0.000,C 90.000,E1 170.443} C_DIS
LIN {X 0.091,Y -378.675,Z 817.735,A 0.000,B 0.000,C 90.000,E1 168.229} C_DIS
LIN {X -0.032,Y -376.346,Z 817.719,A 0.000,B 0.000,C 90.000,E1 165.338} C_DIS
LIN {X -0.174,Y -373.755,Z 817.680,A 0.000,B 0.000,C 90.000,E1 158.411} C_DIS
LIN {X 0.065,Y -374.311,Z 817.668,A 0.000,B 0.000,C 90.000,E1 156.177} C_DIS
LIN {X 0.005,Y -375.642,Z 817.658,A 0.000,B 0.000,C 90.000,E1 154.357} C_DIS
LIN {X 0.044,Y -376.884,Z 817.651,A 0.000,B 0.000,C 90.000,E1 153.256} C_DIS
LIN {X 0.104,Y -378.622,Z 817.645,A 0.000,B 0.000,C 90.000,E1 152.153} C_DIS
LIN {X 0.045,Y -380.053,Z 817.641,A 0.000,B 0.000,C 90.000,E1 151.435} C_DIS
LIN {X -0.001,Y -381.866,Z 817.637,A 0.000,B 0.000,C 90.000,E1 150.717} C_DIS
LIN {X 0.018,Y -385.666,Z 817.630,A 0.000,B 0.000,C 90.000,E1 149.459} C_DIS
LIN {X 0.029,Y -387.932,Z 817.627,A 0.000,B 0.000,C 90.000,E1 148.918} C_DIS
LIN {X 0.073,Y -390.421,Z 817.625,A 0.000,B 0.000,C 90.000,E1 148.408} C_DIS
LIN {X -0.123,Y -394.235,Z 817.621,A 0.000,B 0.000,C 90.000,E1 147.788} C_DIS
LIN {X -0.061,Y -397.744,Z 817.618,A 0.000,B 0.000,C 90.000,E1 147.248} C_DIS
LIN {X 0.041,Y -408.167,Z 817.612,A 0.000,B 0.000,C 90.000,E1 146.087} C_DIS
LIN {X -0.115,Y -411.450,Z 817.610,A 0.000,B 0.000,C 90.000,E1 145.801} C_DIS
LIN {X -0.157,Y -422.816,Z 817.605,A 0.000,B 0.000,C 90.000,E1 144.895} C_DIS
LIN {X 0.006,Y -430.662,Z 817.602,A 0.000,B 0.000,C 90.000,E1 144.322} C_DIS
LIN {X -0.234,Y -435.504,Z 817.600,A 0.000,B 0.000,C 90.000,E1 143.989} C_DIS
LIN {X 0.101,Y -442.988,Z 817.596,A 0.000,B 0.000,C 90.000,E1 143.336} C_DIS
LIN {X -0.191,Y -448.740,Z 817.594,A 0.000,B 0.000,C 90.000,E1 142.844} C_DIS
LIN {X 0.011,Y -453.009,Z 817.591,A 0.000,B 0.000,C 90.000,E1 142.396} C_DIS
LIN {X -0.117,Y -458.403,Z 817.588,A 0.000,B 0.000,C 90.000,E1 141.823} C_DIS
LIN {X 0.090,Y -462.225,Z 817.585,A 0.000,B 0.000,C 90.000,E1 141.331} C_DIS
LIN {X 0.122,Y -464.723,Z 817.583,A 0.000,B 0.000,C 90.000,E1 141.009} C_DIS
LIN {X -0.020,Y -468.570,Z 817.581,A 0.000,B 0.000,C 90.000,E1 140.561} C_DIS
LIN {X 0.104,Y -471.048,Z 817.579,A 0.000,B 0.000,C 90.000,E1 140.231} C_DIS
LIN {X 0.098,Y -478.907,Z 817.573,A 0.000,B 0.000,C 90.000,E1 139.138} C_DIS
LIN {X 0.011,Y -483.036,Z 817.570,A 0.000,B 0.000,C 90.000,E1 138.528} C_DIS
LIN {X -0.232,Y -488.637,Z 817.565,A 0.000,B 0.000,C 90.000,E1 137.634} C_DIS
LIN {X -0.001,Y -491.268,Z 817.562,A 0.000,B 0.000,C 90.000,E1 137.148} C_DIS
LIN {X -0.243,Y -498.686,Z 817.554,A 0.000,B 0.000,C 90.000,E1 135.810} C_DIS
LIN {X -0.235,Y -504.238,Z 817.549,A 0.000,B 0.000,C 90.000,E1 134.757} C_DIS
LIN {X 0.329,Y -508.015,Z 817.544,A 0.000,B 0.000,C 90.000,E1 133.947} C_DIS
LIN {X 0.109,Y -513.187,Z 817.539,A 0.000,B 0.000,C 90.000,E1 132.933} C_DIS
LIN {X -0.101,Y -516.048,Z 817.535,A 0.000,B 0.000,C 90.000,E1 132.366} C_DIS
LIN {X 0.089,Y -518.567,Z 817.532,A 0.000,B 0.000,C 90.000,E1 131.757} C_DIS
LIN {X -0.152,Y -522.065,Z 817.527,A 0.000,B 0.000,C 90.000,E1 130.906} C_DIS
LIN {X 0.080,Y -524.242,Z 817.524,A 0.000,B 0.000,C 90.000,E1 130.297} C_DIS
LIN {X 0.232,Y -529.358,Z 817.516,A 0.000,B 0.000,C 90.000,E1 128.830} C_DIS
LIN {X -0.260,Y -532.685,Z 817.510,A 0.000,B 0.000,C 90.000,E1 127.729} C_DIS
LIN {X -0.285,Y -535.830,Z 817.503,A 0.000,B 0.000,C 90.000,E1 126.583} C_DIS
LIN {X 0.162,Y -537.959,Z 817.498,A 0.000,B 0.000,C 90.000,E1 125.678} C_DIS
LIN {X 0.196,Y -539.304,Z 817.494,A 0.000,B 0.000,C 90.000,E1 124.818} C_DIS
LIN {X -0.081,Y -539.984,Z 817.490,A 0.000,B 0.000,C 90.000,E1 124.278} C_DIS
LIN {X -0.034,Y -540.545,Z 817.486,A 0.000,B 0.000,C 90.000,E1 123.420} C_DIS
LIN {X -0.056,Y -542.489,Z 817.479,A 0.000,B 0.000,C 90.000,E1 122.291} C_DIS
LIN {X -0.038,Y -543.136,Z 817.478,A 0.000,B 0.000,C 90.000,E1 122.005} C_DIS
LIN {X 0.096,Y -543.775,Z 817.477,A 0.000,B 0.000,C 90.000,E1 121.799} C_DIS
LIN {X -0.169,Y -544.502,Z 817.475,A 0.000,B 0.000,C 90.000,E1 121.544} C_DIS
LIN {X -0.149,Y -545.072,Z 817.474,A 0.000,B 0.000,C 90.000,E1 121.258} C_DIS
LIN {X -0.326,Y -545.853,Z 817.472,A 0.000,B 0.000,C 90.000,E1 121.003} C_DIS
LIN {X -0.086,Y -547.149,Z 817.469,A 0.000,B 0.000,C 90.000,E1 120.413} C_DIS
LIN {X 0.003,Y -547.928,Z 817.467,A 0.000,B 0.000,C 90.000,E1 120.129} C_DIS
LIN {X 0.260,Y -549.033,Z 817.464,A 0.000,B 0.000,C 90.000,E1 119.539} C_DIS
LIN {X 0.045,Y -550.400,Z 817.461,A 0.000,B 0.000,C 90.000,E1 118.999} C_DIS
LIN {X 0.056,Y -551.601,Z 817.458,A 0.000,B 0.000,C 90.000,E1 118.437} C_DIS
LIN {X -0.110,Y -554.020,Z 817.452,A 0.000,B 0.000,C 90.000,E1 117.334} C_DIS
LIN {X -0.247,Y -556.025,Z 817.446,A 0.000,B 0.000,C 90.000,E1 116.232} C_DIS
LIN {X 0.350,Y -557.256,Z 817.441,A 0.000,B 0.000,C 90.000,E1 115.335} C_DIS
LIN {X 0.305,Y -559.026,Z 817.433,A 0.000,B 0.000,C 90.000,E1 113.951} C_DIS
LIN {X 0.070,Y -560.643,Z 817.426,A 0.000,B 0.000,C 90.000,E1 112.589} C_DIS
LIN {X -0.135,Y -561.939,Z 817.418,A 0.000,B 0.000,C 90.000,E1 111.227} C_DIS
LIN {X -0.118,Y -562.545,Z 817.412,A 0.000,B 0.000,C 90.000,E1 110.120} C_DIS
LIN {X 0.114,Y -562.794,Z 817.407,A 0.000,B 0.000,C 90.000,E1 109.268} C_DIS
LIN {X -0.049,Y -563.048,Z 817.401,A 0.000,B 0.000,C 90.000,E1 108.181} C_DIS
LIN {X -0.144,Y -563.427,Z 817.390,A 0.000,B 0.000,C 90.000,E1 106.260} C_DIS
LIN {X -0.163,Y -564.747,Z 817.373,A 0.000,B 0.000,C 90.000,E1 103.231} C_DIS
LIN {X 0.065,Y -566.153,Z 817.361,A 0.000,B 0.000,C 90.000,E1 101.007} C_DIS
LIN {X -0.037,Y -567.555,Z 817.351,A 0.000,B 0.000,C 90.000,E1 99.095} C_DIS
LIN {X 0.195,Y -568.503,Z 817.343,A 0.000,B 0.000,C 90.000,E1 97.701} C_DIS
LIN {X -0.096,Y -569.500,Z 817.334,A 0.000,B 0.000,C 90.000,E1 96.087} C_DIS
LIN {X -0.206,Y -569.944,Z 817.329,A 0.000,B 0.000,C 90.000,E1 95.277} C_DIS
LIN {X -0.079,Y -570.585,Z 817.322,A 0.000,B 0.000,C 90.000,E1 93.898} C_DIS
LIN {X 0.155,Y -571.213,Z 817.313,A 0.000,B 0.000,C 90.000,E1 92.236} C_DIS
LIN {X 0.273,Y -571.707,Z 817.305,A 0.000,B 0.000,C 90.000,E1 90.859} C_DIS
LIN {X -0.186,Y -572.104,Z 817.297,A 0.000,B 0.000,C 90.000,E1 89.542} C_DIS
LIN {X 0.085,Y -572.553,Z 817.288,A 0.000,B 0.000,C 90.000,E1 87.879} C_DIS
LIN {X 0.093,Y -572.817,Z 817.282,A 0.000,B 0.000,C 90.000,E1 86.788} C_DIS
LIN {X -0.026,Y -573.212,Z 817.272,A 0.000,B 0.000,C 90.000,E1 84.894} C_DIS
LIN {X -0.223,Y -573.468,Z 817.263,A 0.000,B 0.000,C 90.000,E1 83.280} C_DIS
LIN {X 0.030,Y -573.792,Z 817.255,A 0.000,B 0.000,C 90.000,E1 81.894} C_DIS
LIN {X 0.113,Y -574.299,Z 817.244,A 0.000,B 0.000,C 90.000,E1 79.982} C_DIS
LIN {X 0.208,Y -574.667,Z 817.235,A 0.000,B 0.000,C 90.000,E1 78.342} C_DIS
LIN {X 0.113,Y -574.909,Z 817.228,A 0.000,B 0.000,C 90.000,E1 76.992} C_DIS
LIN {X 0.213,Y -574.998,Z 817.219,A 0.000,B 0.000,C 90.000,E1 75.353} C_DIS
LIN {X 0.044,Y -574.974,Z 817.210,A 0.000,B 0.000,C 90.000,E1 73.740} C_DIS
LIN {X 0.238,Y -574.853,Z 817.202,A 0.000,B 0.000,C 90.000,E1 72.362} C_DIS
LIN {X 0.243,Y -574.616,Z 817.193,A 0.000,B 0.000,C 90.000,E1 70.732} C_DIS
LIN {X 0.068,Y -574.294,Z 817.186,A 0.000,B 0.000,C 90.000,E1 69.390} C_DIS
LIN {X 0.259,Y -573.997,Z 817.180,A 0.000,B 0.000,C 90.000,E1 68.284} C_DIS
LIN {X -0.087,Y -573.637,Z 817.174,A 0.000,B 0.000,C 90.000,E1 67.230} C_DIS
LIN {X -0.079,Y -573.060,Z 817.166,A 0.000,B 0.000,C 90.000,E1 65.869} C_DIS
LIN {X 0.143,Y -572.451,Z 817.158,A 0.000,B 0.000,C 90.000,E1 64.485} C_DIS
LIN {X 0.090,Y -571.684,Z 817.151,A 0.000,B 0.000,C 90.000,E1 63.127} C_DIS
LIN {X 0.198,Y -570.875,Z 817.145,A 0.000,B 0.000,C 90.000,E1 62.025} C_DIS
LIN {X 0.295,Y -569.908,Z 817.139,A 0.000,B 0.000,C 90.000,E1 60.923} C_DIS
LIN {X -0.124,Y -568.721,Z 817.133,A 0.000,B 0.000,C 90.000,E1 59.871} C_DIS
LIN {X 0.217,Y -567.347,Z 817.127,A 0.000,B 0.000,C 90.000,E1 58.742} C_DIS
LIN {X 0.159,Y -565.352,Z 817.119,A 0.000,B 0.000,C 90.000,E1 57.375} C_DIS
LIN {X -0.033,Y -563.469,Z 817.113,A 0.000,B 0.000,C 90.000,E1 56.294} C_DIS
LIN {X 0.057,Y -561.238,Z 817.107,A 0.000,B 0.000,C 90.000,E1 55.182} C_DIS
LIN {X 0.112,Y -558.803,Z 817.101,A 0.000,B 0.000,C 90.000,E1 54.069} C_DIS
LIN {X -0.072,Y -556.672,Z 817.096,A 0.000,B 0.000,C 90.000,E1 53.256} C_DIS
LIN {X 0.172,Y -554.297,Z 817.091,A 0.000,B 0.000,C 90.000,E1 52.396} C_DIS
LIN {X -0.047,Y -551.637,Z 817.087,A 0.000,B 0.000,C 90.000,E1 51.582} C_DIS
LIN {X 0.136,Y -548.619,Z 817.082,A 0.000,B 0.000,C 90.000,E1 50.723} C_DIS
LIN {X -0.185,Y -546.458,Z 817.079,A 0.000,B 0.000,C 90.000,E1 50.194} C_DIS
LIN {X 0.090,Y -543.522,Z 817.075,A 0.000,B 0.000,C 90.000,E1 49.461} C_DIS
LIN {X -0.267,Y -540.996,Z 817.072,A 0.000,B 0.000,C 90.000,E1 48.933} C_DIS
LIN {X -0.277,Y -536.636,Z 817.067,A 0.000,B 0.000,C 90.000,E1 48.081} C_DIS
LIN {X -0.100,Y -534.346,Z 817.065,A 0.000,B 0.000,C 90.000,E1 47.634} C_DIS
LIN {X 0.010,Y -530.018,Z 817.061,A 0.000,B 0.000,C 90.000,E1 46.905} C_DIS
LIN {X 0.303,Y -526.186,Z 817.057,A 0.000,B 0.000,C 90.000,E1 46.296} C_DIS
LIN {X 0.188,Y -521.945,Z 817.054,A 0.000,B 0.000,C 90.000,E1 45.729} C_DIS
LIN {X -0.100,Y -518.642,Z 817.052,A 0.000,B 0.000,C 90.000,E1 45.324} C_DIS
LIN {X -0.265,Y -513.791,Z 817.049,A 0.000,B 0.000,C 90.000,E1 44.757} C_DIS
LIN {X 0.159,Y -509.865,Z 817.046,A 0.000,B 0.000,C 90.000,E1 44.271} C_DIS
LIN {X 0.121,Y -504.469,Z 817.043,A 0.000,B 0.000,C 90.000,E1 43.704} C_DIS
LIN {X -0.112,Y -498.825,Z 817.040,A 0.000,B 0.000,C 90.000,E1 43.176} C_DIS
LIN {X 0.129,Y -493.028,Z 817.037,A 0.000,B 0.000,C 90.000,E1 42.609} C_DIS
LIN {X 0.204,Y -486.940,Z 817.034,A 0.000,B 0.000,C 90.000,E1 42.081} C_DIS
LIN {X 0.101,Y -480.751,Z 817.031,A 0.000,B 0.000,C 90.000,E1 41.595} C_DIS
LIN {X 0.027,Y -471.509,Z 817.027,A 0.000,B 0.000,C 90.000,E1 40.906} C_DIS
LIN {X -0.039,Y -463.519,Z 817.024,A 0.000,B 0.000,C 90.000,E1 40.334} C_DIS
LIN {X 0.136,Y -449.239,Z 817.018,A 0.000,B 0.000,C 90.000,E1 39.277} C_DIS
LIN {X 0.018,Y -420.977,Z 817.006,A 0.000,B 0.000,C 90.000,E1 37.156} C_DIS
LIN {X -0.108,Y -408.787,Z 817.001,A 0.000,B 0.000,C 90.000,E1 36.137} C_DIS
LIN {X -0.209,Y -403.015,Z 816.998,A 0.000,B 0.000,C 90.000,E1 35.598} C_DIS
LIN {X 0.202,Y -400.491,Z 816.996,A 0.000,B 0.000,C 90.000,E1 35.231} C_DIS
LIN {X 0.177,Y -398.892,Z 816.995,A 0.000,B 0.000,C 90.000,E1 35.025} C_DIS
LIN {X 0.139,Y -398.849,Z 816.995,A 0.000,B 0.000,C 90.000,E1 35.025} C_DIS
LIN {X 0.033,Y -393.929,Z 816.977,A 0.000,B 0.000,C 90.000,E1 31.926} C_DIS
LIN {X -0.172,Y -392.811,Z 816.974,A 0.000,B 0.000,C 90.000,E1 31.337} C_DIS
LIN {X -0.005,Y -393.891,Z 816.960,A 0.000,B 0.000,C 90.000,E1 28.743} C_DIS
LIN {X -0.080,Y -395.518,Z 816.944,A 0.000,B 0.000,C 90.000,E1 25.924} C_DIS
LIN {X 0.088,Y -397.461,Z 816.928,A 0.000,B 0.000,C 90.000,E1 23.078} C_DIS
LIN {X -0.156,Y -399.745,Z 816.913,A 0.000,B 0.000,C 90.000,E1 20.301} C_DIS
LIN {X -0.069,Y -403.882,Z 816.891,A 0.000,B 0.000,C 90.000,E1 16.441} C_DIS
LIN {X 0.144,Y -408.755,Z 816.872,A 0.000,B 0.000,C 90.000,E1 12.939} C_DIS
LIN {X -0.034,Y -412.201,Z 816.861,A 0.000,B 0.000,C 90.000,E1 10.894} C_DIS
LIN {X -0.154,Y -416.361,Z 816.847,A 0.000,B 0.000,C 90.000,E1 8.511} C_DIS
LIN {X 0.124,Y -420.081,Z 816.836,A 0.000,B 0.000,C 90.000,E1 6.429} C_DIS
LIN {X -0.052,Y -423.194,Z 816.826,A 0.000,B 0.000,C 90.000,E1 4.759} C_DIS
LIN {X -0.096,Y -427.720,Z 816.813,A 0.000,B 0.000,C 90.000,E1 2.407} C_DIS
LIN {X 0.164,Y -433.160,Z 816.799,A 0.000,B 0.000,C 90.000,E1 359.771} C_DIS
LIN {X -0.141,Y -437.580,Z 816.788,A 0.000,B 0.000,C 90.000,E1 357.822} C_DIS
LIN {X -0.026,Y -441.520,Z 816.779,A 0.000,B 0.000,C 90.000,E1 356.159} C_DIS
LIN {X -0.091,Y -446.336,Z 816.768,A 0.000,B 0.000,C 90.000,E1 354.204} C_DIS
LIN {X -0.186,Y -450.488,Z 816.759,A 0.000,B 0.000,C 90.000,E1 352.591} C_DIS
LIN {X -0.146,Y -454.784,Z 816.750,A 0.000,B 0.000,C 90.000,E1 350.971} C_DIS
LIN {X 0.066,Y -455.791,Z 816.748,A 0.000,B 0.000,C 90.000,E1 350.622} C_DIS
LIN {X -0.018,Y -457.593,Z 816.745,A 0.000,B 0.000,C 90.000,E1 350.151} C_DIS
LIN {X -0.001,Y -459.483,Z 816.743,A 0.000,B 0.000,C 90.000,E1 349.803} C_DIS
LIN {X 0.074,Y -460.430,Z 816.742,A 0.000,B 0.000,C 90.000,E1 349.634} C_DIS
LIN {X 0.000,Y -463.174,Z 816.741,A 0.000,B 0.000,C 90.000,E1 349.285} C_DIS
LIN {X -0.113,Y -469.612,Z 816.737,A 0.000,B 0.000,C 90.000,E1 348.701} C_DIS
LIN {X -0.015,Y -473.447,Z 816.736,A 0.000,B 0.000,C 90.000,E1 348.409} C_DIS
LIN {X 0.018,Y -476.533,Z 816.734,A 0.000,B 0.000,C 90.000,E1 348.173} C_DIS
LIN {X -0.170,Y -489.406,Z 816.730,A 0.000,B 0.000,C 90.000,E1 347.353} C_DIS
LIN {X 0.157,Y -498.802,Z 816.726,A 0.000,B 0.000,C 90.000,E1 346.700} C_DIS
LIN {X -0.066,Y -511.520,Z 816.722,A 0.000,B 0.000,C 90.000,E1 345.880} C_DIS
LIN {X 0.198,Y -523.955,Z 816.717,A 0.000,B 0.000,C 90.000,E1 344.991} C_DIS
LIN {X -0.130,Y -534.696,Z 816.713,A 0.000,B 0.000,C 90.000,E1 344.267} C_DIS
LIN {X 0.147,Y -543.551,Z 816.709,A 0.000,B 0.000,C 90.000,E1 343.559} C_DIS
LIN {X -0.249,Y -553.641,Z 816.704,A 0.000,B 0.000,C 90.000,E1 342.779} C_DIS
LIN {X 0.322,Y -559.192,Z 816.702,A 0.000,B 0.000,C 90.000,E1 342.236} C_DIS
LIN {X 0.064,Y -565.738,Z 816.698,A 0.000,B 0.000,C 90.000,E1 341.638} C_DIS
LIN {X 0.273,Y -570.824,Z 816.695,A 0.000,B 0.000,C 90.000,E1 341.094} C_DIS
LIN {X 0.276,Y -576.970,Z 816.691,A 0.000,B 0.000,C 90.000,E1 340.423} C_DIS
LIN {X 0.215,Y -582.495,Z 816.688,A 0.000,B 0.000,C 90.000,E1 339.752} C_DIS
LIN {X 0.270,Y -586.533,Z 816.685,A 0.000,B 0.000,C 90.000,E1 339.209} C_DIS
LIN {X 0.230,Y -592.169,Z 816.680,A 0.000,B 0.000,C 90.000,E1 338.411} C_DIS
LIN {X -0.257,Y -596.442,Z 816.677,A 0.000,B 0.000,C 90.000,E1 337.794} C_DIS
LIN {X -0.281,Y -602.930,Z 816.671,A 0.000,B 0.000,C 90.000,E1 336.741} C_DIS
LIN {X 0.051,Y -608.325,Z 816.666,A 0.000,B 0.000,C 90.000,E1 335.793} C_DIS
LIN {X -0.387,Y -615.065,Z 816.659,A 0.000,B 0.000,C 90.000,E1 334.665} C_DIS
LIN {X 0.104,Y -619.273,Z 816.655,A 0.000,B 0.000,C 90.000,E1 333.845} C_DIS
LIN {X 0.092,Y -625.969,Z 816.648,A 0.000,B 0.000,C 90.000,E1 332.564} C_DIS
LIN {X -0.112,Y -630.258,Z 816.643,A 0.000,B 0.000,C 90.000,E1 331.691} C_DIS
LIN {X 0.010,Y -634.979,Z 816.637,A 0.000,B 0.000,C 90.000,E1 330.667} C_DIS
LIN {X -0.008,Y -640.650,Z 816.630,A 0.000,B 0.000,C 90.000,E1 329.410} C_DIS
LIN {X 0.001,Y -644.759,Z 816.625,A 0.000,B 0.000,C 90.000,E1 328.408} C_DIS
LIN {X 0.059,Y -648.618,Z 816.619,A 0.000,B 0.000,C 90.000,E1 327.406} C_DIS
LIN {X 0.441,Y -651.283,Z 816.615,A 0.000,B 0.000,C 90.000,E1 326.628} C_DIS
LIN {X 0.037,Y -654.601,Z 816.609,A 0.000,B 0.000,C 90.000,E1 325.674} C_DIS
LIN {X 0.042,Y -657.690,Z 816.604,A 0.000,B 0.000,C 90.000,E1 324.689} C_DIS
LIN {X -0.357,Y -661.319,Z 816.597,A 0.000,B 0.000,C 90.000,E1 323.497} C_DIS
LIN {X 0.168,Y -663.350,Z 816.593,A 0.000,B 0.000,C 90.000,E1 322.718} C_DIS
LIN {X 0.162,Y -665.759,Z 816.588,A 0.000,B 0.000,C 90.000,E1 321.743} C_DIS
LIN {X 0.284,Y -668.588,Z 816.581,A 0.000,B 0.000,C 90.000,E1 320.517} C_DIS
LIN {X 0.358,Y -671.140,Z 816.574,A 0.000,B 0.000,C 90.000,E1 319.299} C_DIS
LIN {X -0.039,Y -673.048,Z 816.569,A 0.000,B 0.000,C 90.000,E1 318.366} C_DIS
LIN {X 0.066,Y -674.450,Z 816.565,A 0.000,B 0.000,C 90.000,E1 317.634} C_DIS
LIN {X -0.268,Y -676.382,Z 816.558,A 0.000,B 0.000,C 90.000,E1 316.458} C_DIS
LIN {X -0.136,Y -677.834,Z 816.553,A 0.000,B 0.000,C 90.000,E1 315.486} C_DIS
LIN {X -0.022,Y -678.822,Z 816.549,A 0.000,B 0.000,C 90.000,E1 314.757} C_DIS
LIN {X 0.186,Y -680.356,Z 816.542,A 0.000,B 0.000,C 90.000,E1 313.542} C_DIS
LIN {X 0.034,Y -682.339,Z 816.533,A 0.000,B 0.000,C 90.000,E1 311.881} C_DIS
LIN {X -0.122,Y -683.657,Z 816.526,A 0.000,B 0.000,C 90.000,E1 310.701} C_DIS
LIN {X -0.194,Y -685.133,Z 816.518,A 0.000,B 0.000,C 90.000,E1 309.277} C_DIS
LIN {X 0.291,Y -686.484,Z 816.510,A 0.000,B 0.000,C 90.000,E1 307.810} C_DIS
LIN {X 0.012,Y -687.912,Z 816.501,A 0.000,B 0.000,C 90.000,E1 306.171} C_DIS
LIN {X 0.123,Y -689.034,Z 816.493,A 0.000,B 0.000,C 90.000,E1 304.739} C_DIS
LIN {X 0.422,Y -690.043,Z 816.485,A 0.000,B 0.000,C 90.000,E1 303.293} C_DIS
LIN {X -0.217,Y -691.058,Z 816.477,A 0.000,B 0.000,C 90.000,E1 301.926} C_DIS
LIN {X 0.339,Y -692.144,Z 816.469,A 0.000,B 0.000,C 90.000,E1 300.463} C_DIS
LIN {X -0.027,Y -693.103,Z 816.462,A 0.000,B 0.000,C 90.000,E1 299.077} C_DIS
LIN {X 0.229,Y -694.087,Z 816.454,A 0.000,B 0.000,C 90.000,E1 297.641} C_DIS
LIN {X -0.188,Y -695.330,Z 816.445,A 0.000,B 0.000,C 90.000,E1 296.027} C_DIS
LIN {X 0.152,Y -696.269,Z 816.438,A 0.000,B 0.000,C 90.000,E1 294.823} C_DIS
LIN {X -0.260,Y -696.594,Z 816.435,A 0.000,B 0.000,C 90.000,E1 294.387} C_DIS
LIN {X 0.224,Y -696.427,Z 816.432,A 0.000,B 0.000,C 90.000,E1 293.643} C_DIS
LIN {X -0.184,Y -695.254,Z 816.429,A 0.000,B 0.000,C 90.000,E1 293.206} C_DIS
LIN {X 0.067,Y -694.425,Z 816.428,A 0.000,B 0.000,C 90.000,E1 292.950} C_DIS
LIN {X 0.190,Y -693.720,Z 816.427,A 0.000,B 0.000,C 90.000,E1 292.823} C_DIS
LIN {X 0.167,Y -691.459,Z 816.426,A 0.000,B 0.000,C 90.000,E1 292.589} C_DIS
LIN {X -0.207,Y -689.050,Z 816.424,A 0.000,B 0.000,C 90.000,E1 292.386} C_DIS
LIN {X -0.063,Y -687.648,Z 816.424,A 0.000,B 0.000,C 90.000,E1 292.259} C_DIS
LIN {X -0.086,Y -685.774,Z 816.423,A 0.000,B 0.000,C 90.000,E1 292.153} C_DIS
LIN {X -0.053,Y -681.577,Z 816.422,A 0.000,B 0.000,C 90.000,E1 291.972} C_DIS
LIN {X 0.033,Y -676.093,Z 816.421,A 0.000,B 0.000,C 90.000,E1 291.770} C_DIS
LIN {X -0.032,Y -672.390,Z 816.420,A 0.000,B 0.000,C 90.000,E1 291.663} C_DIS
LIN {X 0.117,Y -662.881,Z 816.419,A 0.000,B 0.000,C 90.000,E1 291.482} C_DIS
LIN {X -0.168,Y -648.557,Z 816.418,A 0.000,B 0.000,C 90.000,E1 291.280} C_DIS
LIN {X -0.169,Y -634.817,Z 816.417,A 0.000,B 0.000,C 90.000,E1 291.025} C_DIS
LIN {X 0.188,Y -623.087,Z 816.415,A 0.000,B 0.000,C 90.000,E1 290.737} C_DIS
LIN {X 0.218,Y -616.691,Z 816.414,A 0.000,B 0.000,C 90.000,E1 290.556} C_DIS
LIN {X 0.221,Y -609.628,Z 816.413,A 0.000,B 0.000,C 90.000,E1 290.301} C_DIS
LIN {X -0.127,Y -607.729,Z 816.412,A 0.000,B 0.000,C 90.000,E1 290.248} C_DIS
LIN {X 0.075,Y -603.253,Z 816.411,A 0.000,B 0.000,C 90.000,E1 289.993} C_DIS
LIN {X 0.181,Y -602.549,Z 816.411,A 0.000,B 0.000,C 90.000,E1 289.939} C_DIS
LIN {X 0.079,Y -601.199,Z 816.410,A 0.000,B 0.000,C 90.000,E1 289.812} C_DIS
LIN {X 0.038,Y -601.178,Z 816.410,A 0.000,B 0.000,C 90.000,E1 289.812} C_DIS
LIN {X 0.106,Y -600.853,Z 816.408,A 0.000,B 0.000,C 90.000,E1 289.504} C_DIS
LIN {X -0.139,Y -600.963,Z 816.408,A 0.000,B 0.000,C 90.000,E1 289.396} C_DIS
LIN {X -0.152,Y -602.648,Z 816.406,A 0.000,B 0.000,C 90.000,E1 289.014} C_DIS
LIN {X 0.088,Y -604.877,Z 816.403,A 0.000,B 0.000,C 90.000,E1 288.598} C_DIS
LIN {X 0.303,Y -608.399,Z 816.401,A 0.000,B 0.000,C 90.000,E1 288.055} C_DIS
LIN {X -0.259,Y -612.103,Z 816.397,A 0.000,B 0.000,C 90.000,E1 287.457} C_DIS
LIN {X 0.073,Y -613.383,Z 816.395,A 0.000,B 0.000,C 90.000,E1 287.166} C_DIS
LIN {X 0.108,Y -616.628,Z 816.391,A 0.000,B 0.000,C 90.000,E1 286.386} C_DIS
LIN {X 0.044,Y -617.626,Z 816.390,A 0.000,B 0.000,C 90.000,E1 286.134} C_DIS
LIN {X -0.055,Y -620.042,Z 816.385,A 0.000,B 0.000,C 90.000,E1 285.371} C_DIS
LIN {X 0.258,Y -621.299,Z 816.383,A 0.000,B 0.000,C 90.000,E1 284.828} C_DIS
LIN {X -0.182,Y -622.268,Z 816.380,A 0.000,B 0.000,C 90.000,E1 284.356} C_DIS
LIN {X 0.204,Y -622.701,Z 816.378,A 0.000,B 0.000,C 90.000,E1 284.064} C_DIS
LIN {X -0.226,Y -623.242,Z 816.375,A 0.000,B 0.000,C 90.000,E1 283.592} C_DIS
LIN {X -0.045,Y -623.524,Z 816.373,A 0.000,B 0.000,C 90.000,E1 283.063} C_DIS
LIN {X -0.257,Y -623.578,Z 816.371,A 0.000,B 0.000,C 90.000,E1 282.827} C_DIS
LIN {X -0.073,Y -623.195,Z 816.368,A 0.000,B 0.000,C 90.000,E1 282.299} C_DIS
LIN {X 0.109,Y -622.500,Z 816.365,A 0.000,B 0.000,C 90.000,E1 281.771} C_DIS
LIN {X 0.285,Y -621.437,Z 816.363,A 0.000,B 0.000,C 90.000,E1 281.243} C_DIS
LIN {X -0.274,Y -620.076,Z 816.360,A 0.000,B 0.000,C 90.000,E1 280.782} C_DIS
LIN {X 0.112,Y -619.311,Z 816.358,A 0.000,B 0.000,C 90.000,E1 280.489} C_DIS
LIN {X 0.265,Y -617.334,Z 816.356,A 0.000,B 0.000,C 90.000,E1 279.962} C_DIS
LIN {X 0.227,Y -614.268,Z 816.352,A 0.000,B 0.000,C 90.000,E1 279.321} C_DIS
LIN {X 0.239,Y -611.316,Z 816.349,A 0.000,B 0.000,C 90.000,E1 278.803} C_DIS
LIN {X 0.320,Y -607.686,Z 816.346,A 0.000,B 0.000,C 90.000,E1 278.276} C_DIS
LIN {X 0.287,Y -603.115,Z 816.343,A 0.000,B 0.000,C 90.000,E1 277.757} C_DIS
LIN {X -0.006,Y -600.264,Z 816.342,A 0.000,B 0.000,C 90.000,E1 277.530} C_DIS
LIN {X -0.086,Y -596.085,Z 816.340,A 0.000,B 0.000,C 90.000,E1 277.182} C_DIS
LIN {X -0.246,Y -589.093,Z 816.338,A 0.000,B 0.000,C 90.000,E1 276.777} C_DIS
LIN {X 0.182,Y -585.166,Z 816.337,A 0.000,B 0.000,C 90.000,E1 276.549} C_DIS
LIN {X 0.073,Y -576.353,Z 816.335,A 0.000,B 0.000,C 90.000,E1 276.201} C_DIS
LIN {X -0.039,Y -574.613,Z 816.334,A 0.000,B 0.000,C 90.000,E1 276.144} C_DIS
LIN {X 0.087,Y -567.599,Z 816.333,A 0.000,B 0.000,C 90.000,E1 275.967} C_DIS
LIN {X -0.102,Y -561.863,Z 816.333,A 0.000,B 0.000,C 90.000,E1 275.967} C_DIS
LIN {X -0.131,Y -553.930,Z 816.333,A 0.000,B 0.000,C 90.000,E1 275.967} C_DIS
LIN {X 0.141,Y -552.188,Z 816.333,A 0.000,B 0.000,C 90.000,E1 275.910} C_DIS
LIN {X 0.098,Y -551.495,Z 816.333,A 0.000,B 0.000,C 90.000,E1 275.853} C_DIS
LIN {X -0.204,Y -550.203,Z 816.331,A 0.000,B 0.000,C 90.000,E1 275.568} C_DIS
LIN {X -0.103,Y -549.857,Z 816.329,A 0.000,B 0.000,C 90.000,E1 275.277} C_DIS
LIN {X -0.165,Y -548.354,Z 816.317,A 0.000,B 0.000,C 90.000,E1 273.037} C_DIS
LIN {X 0.133,Y -547.195,Z 816.307,A 0.000,B 0.000,C 90.000,E1 271.318} C_DIS
LIN {X -0.235,Y -546.397,Z 816.301,A 0.000,B 0.000,C 90.000,E1 270.229} C_DIS
LIN {X 0.013,Y -545.236,Z 816.292,A 0.000,B 0.000,C 90.000,E1 268.511} C_DIS
LIN {X -0.213,Y -543.700,Z 816.279,A 0.000,B 0.000,C 90.000,E1 266.274} C_DIS
LIN {X -0.008,Y -542.851,Z 816.271,A 0.000,B 0.000,C 90.000,E1 264.837} C_DIS
LIN {X 0.150,Y -542.316,Z 816.267,A 0.000,B 0.000,C 90.000,E1 263.970} C_DIS
LIN {X -0.146,Y -540.852,Z 816.257,A 0.000,B 0.000,C 90.000,E1 262.299} C_DIS
LIN {X 0.119,Y -539.385,Z 816.248,A 0.000,B 0.000,C 90.000,E1 260.566} C_DIS
LIN {X -0.069,Y -537.963,Z 816.240,A 0.000,B 0.000,C 90.000,E1 259.162} C_DIS
LIN {X 0.254,Y -536.554,Z 816.232,A 0.000,B 0.000,C 90.000,E1 257.701} C_DIS
LIN {X 0.017,Y -535.096,Z 816.224,A 0.000,B 0.000,C 90.000,E1 256.297} C_DIS
LIN {X 0.056,Y -533.154,Z 816.214,A 0.000,B 0.000,C 90.000,E1 254.574} C_DIS
LIN {X 0.052,Y -531.179,Z 816.205,A 0.000,B 0.000,C 90.000,E1 252.851} C_DIS
LIN {X 0.136,Y -529.430,Z 816.197,A 0.000,B 0.000,C 90.000,E1 251.402} C_DIS
LIN {X 0.188,Y -527.979,Z 816.190,A 0.000,B 0.000,C 90.000,E1 250.242} C_DIS
LIN {X 0.220,Y -526.383,Z 816.184,A 0.000,B 0.000,C 90.000,E1 249.082} C_DIS
LIN {X -0.261,Y -524.727,Z 816.178,A 0.000,B 0.000,C 90.000,E1 247.975} C_DIS
LIN {X -0.083,Y -523.062,Z 816.171,A 0.000,B 0.000,C 90.000,E1 246.794} C_DIS
LIN {X -0.257,Y -520.845,Z 816.163,A 0.000,B 0.000,C 90.000,E1 245.357} C_DIS
LIN {X 0.073,Y -518.931,Z 816.156,A 0.000,B 0.000,C 90.000,E1 244.152} C_DIS
LIN {X 0.034,Y -516.466,Z 816.148,A 0.000,B 0.000,C 90.000,E1 242.692} C_DIS
LIN {X -0.042,Y -514.952,Z 816.143,A 0.000,B 0.000,C 90.000,E1 241.820} C_DIS
LIN {X -0.018,Y -511.625,Z 816.134,A 0.000,B 0.000,C 90.000,E1 240.049} C_DIS
LIN {X -0.050,Y -509.446,Z 816.127,A 0.000,B 0.000,C 90.000,E1 238.869} C_DIS
LIN {X -0.185,Y -507.694,Z 816.122,A 0.000,B 0.000,C 90.000,E1 237.995} C_DIS
LIN {X -0.023,Y -505.222,Z 816.116,A 0.000,B 0.000,C 90.000,E1 236.786} C_DIS
LIN {X -0.156,Y -501.973,Z 816.107,A 0.000,B 0.000,C 90.000,E1 235.308} C_DIS
LIN {X -0.216,Y -499.218,Z 816.101,A 0.000,B 0.000,C 90.000,E1 234.116} C_DIS
LIN {X -0.191,Y -497.084,Z 816.096,A 0.000,B 0.000,C 90.000,E1 233.210} C_DIS
LIN {X -0.176,Y -493.407,Z 816.087,A 0.000,B 0.000,C 90.000,E1 231.698} C_DIS
LIN {X 0.214,Y -487.583,Z 816.074,A 0.000,B 0.000,C 90.000,E1 229.218} C_DIS
LIN {X 0.160,Y -484.816,Z 816.067,A 0.000,B 0.000,C 90.000,E1 228.000} C_DIS
LIN {X -0.229,Y -480.001,Z 816.055,A 0.000,B 0.000,C 90.000,E1 225.891} C_DIS
LIN {X -0.190,Y -475.895,Z 816.044,A 0.000,B 0.000,C 90.000,E1 224.028} C_DIS
LIN {X -0.002,Y -472.581,Z 816.036,A 0.000,B 0.000,C 90.000,E1 222.447} C_DIS
LIN {X -0.002,Y -467.946,Z 816.024,A 0.000,B 0.000,C 90.000,E1 220.253} C_DIS
LIN {X 0.229,Y -463.374,Z 816.011,A 0.000,B 0.000,C 90.000,E1 218.016} C_DIS
LIN {X 0.012,Y -459.425,Z 816.001,A 0.000,B 0.000,C 90.000,E1 216.137} C_DIS
LIN {X -0.029,Y -456.743,Z 815.994,A 0.000,B 0.000,C 90.000,E1 214.865} C_DIS
LIN {X -0.093,Y -454.745,Z 815.988,A 0.000,B 0.000,C 90.000,E1 213.913} C_DIS
LIN {X -0.079,Y -452.062,Z 815.981,A 0.000,B 0.000,C 90.000,E1 212.625} C_DIS
LIN {X 0.106,Y -450.774,Z 815.978,A 0.000,B 0.000,C 90.000,E1 211.957} C_DIS
LIN {X 0.212,Y -446.769,Z 815.967,A 0.000,B 0.000,C 90.000,E1 210.001} C_DIS
LIN {X -0.129,Y -444.194,Z 815.960,A 0.000,B 0.000,C 90.000,E1 208.743} C_DIS
LIN {X 0.113,Y -441.013,Z 815.951,A 0.000,B 0.000,C 90.000,E1 207.078} C_DIS
LIN {X -0.129,Y -438.482,Z 815.943,A 0.000,B 0.000,C 90.000,E1 205.796} C_DIS
LIN {X -0.004,Y -435.175,Z 815.934,A 0.000,B 0.000,C 90.000,E1 204.131} C_DIS
LIN {X -0.089,Y -431.297,Z 815.923,A 0.000,B 0.000,C 90.000,E1 202.153} C_DIS
LIN {X -0.058,Y -426.804,Z 815.910,A 0.000,B 0.000,C 90.000,E1 199.812} C_DIS
LIN {X -0.074,Y -424.177,Z 815.903,A 0.000,B 0.000,C 90.000,E1 198.471} C_DIS
LIN {X -0.034,Y -420.263,Z 815.891,A 0.000,B 0.000,C 90.000,E1 196.441} C_DIS
LIN {X -0.088,Y -416.359,Z 815.880,A 0.000,B 0.000,C 90.000,E1 194.411} C_DIS
LIN {X -0.006,Y -411.868,Z 815.867,A 0.000,B 0.000,C 90.000,E1 192.007} C_DIS
LIN {X -0.172,Y -408.616,Z 815.857,A 0.000,B 0.000,C 90.000,E1 190.310} C_DIS
LIN {X -0.078,Y -405.381,Z 815.848,A 0.000,B 0.000,C 90.000,E1 188.568} C_DIS
LIN {X -0.115,Y -401.483,Z 815.836,A 0.000,B 0.000,C 90.000,E1 186.486} C_DIS
LIN {X 0.035,Y -397.232,Z 815.822,A 0.000,B 0.000,C 90.000,E1 184.012} C_DIS
LIN {X -0.057,Y -393.096,Z 815.807,A 0.000,B 0.000,C 90.000,E1 181.203} C_DIS
LIN {X 0.183,Y -389.905,Z 815.793,A 0.000,B 0.000,C 90.000,E1 178.682} C_DIS
LIN {X 0.063,Y -387.462,Z 815.781,A 0.000,B 0.000,C 90.000,E1 176.560} C_DIS
LIN {X 0.106,Y -384.183,Z 815.765,A 0.000,B 0.000,C 90.000,E1 173.685} C_DIS
LIN {X -0.124,Y -381.607,Z 815.751,A 0.000,B 0.000,C 90.000,E1 171.197} C_DIS
LIN {X -0.092,Y -380.236,Z 815.743,A 0.000,B 0.000,C 90.000,E1 169.746} C_DIS
LIN {X -0.017,Y -378.986,Z 815.735,A 0.000,B 0.000,C 90.000,E1 168.285} C_DIS
LIN {X -0.220,Y -376.648,Z 815.719,A 0.000,B 0.000,C 90.000,E1 165.408} C_DIS
LIN {X 0.069,Y -374.435,Z 815.696,A 0.000,B 0.000,C 90.000,E1 161.348} C_DIS
LIN {X -0.063,Y -374.214,Z 815.672,A 0.000,B 0.000,C 90.000,E1 156.975} C_DIS
LIN {X 0.104,Y -374.879,Z 815.664,A 0.000,B 0.000,C 90.000,E1 155.485} C_DIS
LIN {X -0.030,Y -375.665,Z 815.658,A 0.000,B 0.000,C 90.000,E1 154.409} C_DIS
LIN {X 0.011,Y -376.709,Z 815.652,A 0.000,B 0.000,C 90.000,E1 153.307} C_DIS
LIN {X 0.029,Y -378.852,Z 815.644,A 0.000,B 0.000,C 90.000,E1 151.847} C_DIS
LIN {X -0.030,Y -380.196,Z 815.640,A 0.000,B 0.000,C 90.000,E1 151.129} C_DIS
LIN {X 0.076,Y -383.909,Z 815.632,A 0.000,B 0.000,C 90.000,E1 149.665} C_DIS
LIN {X 0.056,Y -386.409,Z 815.628,A 0.000,B 0.000,C 90.000,E1 148.948} C_DIS
LIN {X 0.087,Y -388.473,Z 815.625,A 0.000,B 0.000,C 90.000,E1 148.456} C_DIS
LIN {X 0.087,Y -390.970,Z 815.622,A 0.000,B 0.000,C 90.000,E1 147.946} C_DIS
LIN {X -0.204,Y -394.015,Z 815.619,A 0.000,B 0.000,C 90.000,E1 147.454} C_DIS
LIN {X -0.020,Y -397.230,Z 815.617,A 0.000,B 0.000,C 90.000,E1 146.962} C_DIS
LIN {X 0.137,Y -399.583,Z 815.615,A 0.000,B 0.000,C 90.000,E1 146.628} C_DIS
LIN {X -0.202,Y -400.669,Z 815.614,A 0.000,B 0.000,C 90.000,E1 146.501} C_DIS
LIN {X 0.274,Y -403.985,Z 815.611,A 0.000,B 0.000,C 90.000,E1 146.008} C_DIS
LIN {X 0.237,Y -407.949,Z 815.609,A 0.000,B 0.000,C 90.000,E1 145.595} C_DIS
LIN {X 0.077,Y -415.345,Z 815.605,A 0.000,B 0.000,C 90.000,E1 144.895} C_DIS
LIN {X -0.199,Y -431.501,Z 815.598,A 0.000,B 0.000,C 90.000,E1 143.623} C_DIS
LIN {X -0.137,Y -439.123,Z 815.594,A 0.000,B 0.000,C 90.000,E1 142.970} C_DIS
LIN {X 0.047,Y -444.909,Z 815.591,A 0.000,B 0.000,C 90.000,E1 142.396} C_DIS
LIN {X -0.047,Y -449.163,Z 815.589,A 0.000,B 0.000,C 90.000,E1 141.984} C_DIS
LIN {X 0.041,Y -453.367,Z 815.586,A 0.000,B 0.000,C 90.000,E1 141.537} C_DIS
LIN {X -0.014,Y -458.544,Z 815.583,A 0.000,B 0.000,C 90.000,E1 140.928} C_DIS
LIN {X -0.119,Y -467.165,Z 815.577,A 0.000,B 0.000,C 90.000,E1 139.828} C_DIS
LIN {X 0.184,Y -475.154,Z 815.571,A 0.000,B 0.000,C 90.000,E1 138.690} C_DIS
LIN {X 0.067,Y -479.343,Z 815.567,A 0.000,B 0.000,C 90.000,E1 138.081} C_DIS
LIN {X 0.044,Y -484.080,Z 815.563,A 0.000,B 0.000,C 90.000,E1 137.310} C_DIS
LIN {X 0.297,Y -490.941,Z 815.556,A 0.000,B 0.000,C 90.000,E1 136.053} C_DIS
LIN {X -0.062,Y -494.172,Z 815.553,A 0.000,B 0.000,C 90.000,E1 135.486} C_DIS
LIN {X 0.298,Y -502.872,Z 815.543,A 0.000,B 0.000,C 90.000,E1 133.785} C_DIS
LIN {X 0.130,Y -508.796,Z 815.537,A 0.000,B 0.000,C 90.000,E1 132.609} C_DIS
LIN {X 0.008,Y -512.179,Z 815.533,A 0.000,B 0.000,C 90.000,E1 131.881} C_DIS
LIN {X 0.085,Y -515.806,Z 815.528,A 0.000,B 0.000,C 90.000,E1 130.987} C_DIS
LIN {X -0.066,Y -518.000,Z 815.525,A 0.000,B 0.000,C 90.000,E1 130.415} C_DIS
LIN {X -0.046,Y -522.192,Z 815.518,A 0.000,B 0.000,C 90.000,E1 129.241} C_DIS
LIN {X -0.189,Y -525.123,Z 815.513,A 0.000,B 0.000,C 90.000,E1 128.382} C_DIS
LIN {X -0.263,Y -526.699,Z 815.510,A 0.000,B 0.000,C 90.000,E1 127.810} C_DIS
LIN {X -0.031,Y -529.622,Z 815.505,A 0.000,B 0.000,C 90.000,E1 126.916} C_DIS
LIN {X 0.338,Y -532.180,Z 815.500,A 0.000,B 0.000,C 90.000,E1 126.011} C_DIS
LIN {X 0.001,Y -534.332,Z 815.496,A 0.000,B 0.000,C 90.000,E1 125.185} C_DIS
LIN {X -0.006,Y -535.278,Z 815.492,A 0.000,B 0.000,C 90.000,E1 124.612} C_DIS
LIN {X -0.010,Y -536.070,Z 815.489,A 0.000,B 0.000,C 90.000,E1 124.040} C_DIS
LIN {X -0.160,Y -536.382,Z 815.488,A 0.000,B 0.000,C 90.000,E1 123.913} C_DIS
LIN {X -0.310,Y -536.887,Z 815.488,A 0.000,B 0.000,C 90.000,E1 123.785} C_DIS
LIN {X 0.141,Y -537.490,Z 815.486,A 0.000,B 0.000,C 90.000,E1 123.452} C_DIS
LIN {X -0.190,Y -537.864,Z 815.484,A 0.000,B 0.000,C 90.000,E1 123.166} C_DIS
LIN {X -0.274,Y -537.859,Z 815.484,A 0.000,B 0.000,C 90.000,E1 123.166} C_DIS
LIN {X -0.315,Y -537.863,Z 815.484,A 0.000,B 0.000,C 90.000,E1 123.166} C_DIS
LIN {X 0.001,Y -538.386,Z 815.484,A 0.000,B 0.000,C 90.000,E1 123.038} C_DIS
LIN {X -0.136,Y -539.890,Z 815.481,A 0.000,B 0.000,C 90.000,E1 122.625} C_DIS
LIN {X -0.053,Y -540.627,Z 815.479,A 0.000,B 0.000,C 90.000,E1 122.260} C_DIS
LIN {X -0.119,Y -541.500,Z 815.478,A 0.000,B 0.000,C 90.000,E1 122.054} C_DIS
LIN {X 0.068,Y -542.422,Z 815.477,A 0.000,B 0.000,C 90.000,E1 121.750} C_DIS
LIN {X -0.162,Y -544.790,Z 815.472,A 0.000,B 0.000,C 90.000,E1 120.924} C_DIS
LIN {X -0.163,Y -547.784,Z 815.465,A 0.000,B 0.000,C 90.000,E1 119.795} C_DIS
LIN {X 0.120,Y -551.251,Z 815.458,A 0.000,B 0.000,C 90.000,E1 118.359} C_DIS
LIN {X 0.174,Y -553.217,Z 815.453,A 0.000,B 0.000,C 90.000,E1 117.513} C_DIS
LIN {X -0.278,Y -554.433,Z 815.450,A 0.000,B 0.000,C 90.000,E1 117.001} C_DIS
LIN {X 0.302,Y -555.988,Z 815.445,A 0.000,B 0.000,C 90.000,E1 116.104} C_DIS
LIN {X 0.157,Y -557.274,Z 815.441,A 0.000,B 0.000,C 90.000,E1 115.283} C_DIS
LIN {X -0.092,Y -559.446,Z 815.431,A 0.000,B 0.000,C 90.000,E1 113.643} C_DIS
LIN {X 0.104,Y -560.738,Z 815.425,A 0.000,B 0.000,C 90.000,E1 112.514} C_DIS
LIN {X 0.102,Y -561.779,Z 815.419,A 0.000,B 0.000,C 90.000,E1 111.408} C_DIS
LIN {X -0.200,Y -562.354,Z 815.414,A 0.000,B 0.000,C 90.000,E1 110.610} C_DIS
LIN {X -0.183,Y -562.849,Z 815.408,A 0.000,B 0.000,C 90.000,E1 109.504} C_DIS
LIN {X -0.211,Y -563.177,Z 815.401,A 0.000,B 0.000,C 90.000,E1 108.127} C_DIS
LIN {X -0.297,Y -563.615,Z 815.390,A 0.000,B 0.000,C 90.000,E1 106.205} C_DIS
LIN {X 0.086,Y -564.831,Z 815.375,A 0.000,B 0.000,C 90.000,E1 103.411} C_DIS
LIN {X -0.231,Y -566.245,Z 815.362,A 0.000,B 0.000,C 90.000,E1 101.243} C_DIS
LIN {X -0.236,Y -567.631,Z 815.352,A 0.000,B 0.000,C 90.000,E1 99.321} C_DIS
LIN {X -0.090,Y -568.615,Z 815.344,A 0.000,B 0.000,C 90.000,E1 97.936} C_DIS
LIN {X -0.025,Y -569.293,Z 815.338,A 0.000,B 0.000,C 90.000,E1 96.834} C_DIS
LIN {X 0.093,Y -570.098,Z 815.330,A 0.000,B 0.000,C 90.000,E1 95.454} C_DIS
LIN {X -0.170,Y -570.882,Z 815.321,A 0.000,B 0.000,C 90.000,E1 93.841} C_DIS
LIN {X 0.073,Y -571.508,Z 815.312,A 0.000,B 0.000,C 90.000,E1 92.178} C_DIS
LIN {X 0.195,Y -572.006,Z 815.305,A 0.000,B 0.000,C 90.000,E1 90.802} C_DIS
LIN {X -0.258,Y -572.419,Z 815.297,A 0.000,B 0.000,C 90.000,E1 89.484} C_DIS
LIN {X 0.019,Y -572.856,Z 815.288,A 0.000,B 0.000,C 90.000,E1 87.822} C_DIS
LIN {X 0.167,Y -573.143,Z 815.280,A 0.000,B 0.000,C 90.000,E1 86.445} C_DIS
LIN {X -0.084,Y -573.529,Z 815.271,A 0.000,B 0.000,C 90.000,E1 84.837} C_DIS
LIN {X 0.104,Y -573.764,Z 815.264,A 0.000,B 0.000,C 90.000,E1 83.457} C_DIS
LIN {X -0.019,Y -574.106,Z 815.255,A 0.000,B 0.000,C 90.000,E1 81.837} C_DIS
LIN {X 0.068,Y -574.593,Z 815.244,A 0.000,B 0.000,C 90.000,E1 79.926} C_DIS
LIN {X -0.040,Y -574.907,Z 815.237,A 0.000,B 0.000,C 90.000,E1 78.578} C_DIS
LIN {X -0.132,Y -575.151,Z 815.229,A 0.000,B 0.000,C 90.000,E1 77.229} C_DIS
LIN {X -0.227,Y -575.214,Z 815.221,A 0.000,B 0.000,C 90.000,E1 75.880} C_DIS
LIN {X 0.168,Y -575.206,Z 815.215,A 0.000,B 0.000,C 90.000,E1 74.755} C_DIS
LIN {X -0.187,Y -575.168,Z 815.208,A 0.000,B 0.000,C 90.000,E1 73.433} C_DIS
LIN {X 0.017,Y -574.999,Z 815.200,A 0.000,B 0.000,C 90.000,E1 72.054} C_DIS
LIN {X 0.205,Y -574.771,Z 815.193,A 0.000,B 0.000,C 90.000,E1 70.678} C_DIS
LIN {X 0.026,Y -574.419,Z 815.185,A 0.000,B 0.000,C 90.000,E1 69.337} C_DIS
LIN {X 0.049,Y -574.006,Z 815.178,A 0.000,B 0.000,C 90.000,E1 67.975} C_DIS
LIN {X -0.296,Y -573.624,Z 815.172,A 0.000,B 0.000,C 90.000,E1 66.922} C_DIS
LIN {X -0.056,Y -573.012,Z 815.164,A 0.000,B 0.000,C 90.000,E1 65.537} C_DIS
LIN {X -0.181,Y -572.501,Z 815.158,A 0.000,B 0.000,C 90.000,E1 64.460} C_DIS
LIN {X 0.030,Y -571.721,Z 815.151,A 0.000,B 0.000,C 90.000,E1 63.076} C_DIS
LIN {X 0.134,Y -570.835,Z 815.144,A 0.000,B 0.000,C 90.000,E1 61.975} C_DIS
LIN {X -0.273,Y -569.821,Z 815.138,A 0.000,B 0.000,C 90.000,E1 60.923} C_DIS
LIN {X 0.086,Y -568.608,Z 815.132,A 0.000,B 0.000,C 90.000,E1 59.793} C_DIS
LIN {X -0.352,Y -567.189,Z 815.126,A 0.000,B 0.000,C 90.000,E1 58.742} C_DIS
LIN {X 0.066,Y -565.127,Z 815.119,A 0.000,B 0.000,C 90.000,E1 57.327} C_DIS
LIN {X 0.177,Y -563.183,Z 815.112,A 0.000,B 0.000,C 90.000,E1 56.215} C_DIS
LIN {X 0.266,Y -560.918,Z 815.106,A 0.000,B 0.000,C 90.000,E1 55.102} C_DIS
LIN {X -0.135,Y -558.375,Z 815.100,A 0.000,B 0.000,C 90.000,E1 54.036} C_DIS
LIN {X -0.203,Y -556.170,Z 815.096,A 0.000,B 0.000,C 90.000,E1 53.210} C_DIS
LIN {X 0.031,Y -553.726,Z 815.091,A 0.000,B 0.000,C 90.000,E1 52.351} C_DIS
LIN {X -0.263,Y -551.991,Z 815.088,A 0.000,B 0.000,C 90.000,E1 51.823} C_DIS
LIN {X -0.077,Y -548.987,Z 815.083,A 0.000,B 0.000,C 90.000,E1 50.964} C_DIS
LIN {X -0.003,Y -545.699,Z 815.078,A 0.000,B 0.000,C 90.000,E1 50.114} C_DIS
LIN {X 0.101,Y -542.035,Z 815.074,A 0.000,B 0.000,C 90.000,E1 49.256} C_DIS
LIN {X -0.099,Y -540.075,Z 815.071,A 0.000,B 0.000,C 90.000,E1 48.852} C_DIS
LIN {X -0.298,Y -536.382,Z 815.067,A 0.000,B 0.000,C 90.000,E1 48.162} C_DIS
LIN {X 0.051,Y -533.208,Z 815.064,A 0.000,B 0.000,C 90.000,E1 47.553} C_DIS
LIN {X -0.016,Y -529.716,Z 815.061,A 0.000,B 0.000,C 90.000,E1 46.986} C_DIS
LIN {X 0.276,Y -525.855,Z 815.058,A 0.000,B 0.000,C 90.000,E1 46.377} C_DIS
LIN {X 0.158,Y -521.579,Z 815.055,A 0.000,B 0.000,C 90.000,E1 45.810} C_DIS
LIN {X 0.010,Y -516.974,Z 815.051,A 0.000,B 0.000,C 90.000,E1 45.243} C_DIS
LIN {X 0.061,Y -513.300,Z 815.049,A 0.000,B 0.000,C 90.000,E1 44.798} C_DIS
LIN {X 0.310,Y -508.021,Z 815.046,A 0.000,B 0.000,C 90.000,E1 44.190} C_DIS
LIN {X -0.015,Y -502.457,Z 815.043,A 0.000,B 0.000,C 90.000,E1 43.662} C_DIS
LIN {X 0.131,Y -496.757,Z 815.040,A 0.000,B 0.000,C 90.000,E1 43.095} C_DIS
LIN {X 0.150,Y -492.371,Z 815.037,A 0.000,B 0.000,C 90.000,E1 42.690} C_DIS
LIN {X -0.075,Y -486.271,Z 815.034,A 0.000,B 0.000,C 90.000,E1 42.204} C_DIS
LIN {X -0.081,Y -478.502,Z 815.031,A 0.000,B 0.000,C 90.000,E1 41.595} C_DIS
LIN {X 0.024,Y -467.734,Z 815.027,A 0.000,B 0.000,C 90.000,E1 40.782} C_DIS
LIN {X -0.046,Y -451.791,Z 815.020,A 0.000,B 0.000,C 90.000,E1 39.644} C_DIS
LIN {X -0.291,Y -426.631,Z 815.010,A 0.000,B 0.000,C 90.000,E1 37.810} C_DIS
LIN {X -0.110,Y -409.531,Z 815.002,A 0.000,B 0.000,C 90.000,E1 36.377} C_DIS
LIN {X 0.107,Y -403.790,Z 814.999,A 0.000,B 0.000,C 90.000,E1 35.804} C_DIS
LIN {X -0.007,Y -401.067,Z 814.997,A 0.000,B 0.000,C 90.000,E1 35.518} C_DIS
LIN {X -0.204,Y -399.282,Z 814.996,A 0.000,B 0.000,C 90.000,E1 35.311} C_DIS
LIN {X -0.231,Y -399.272,Z 814.996,A 0.000,B 0.000,C 90.000,E1 35.311} C_DIS
LIN {X 0.146,Y -393.951,Z 814.978,A 0.000,B 0.000,C 90.000,E1 31.926} C_DIS
LIN {X 0.006,Y -393.012,Z 814.975,A 0.000,B 0.000,C 90.000,E1 31.416} C_DIS
LIN {X 0.115,Y -394.120,Z 814.960,A 0.000,B 0.000,C 90.000,E1 28.743} C_DIS
LIN {X 0.047,Y -395.726,Z 814.944,A 0.000,B 0.000,C 90.000,E1 25.924} C_DIS
LIN {X -0.144,Y -397.665,Z 814.928,A 0.000,B 0.000,C 90.000,E1 23.131} C_DIS
LIN {X -0.092,Y -399.609,Z 814.915,A 0.000,B 0.000,C 90.000,E1 20.663} C_DIS
LIN {X 0.010,Y -403.216,Z 814.895,A 0.000,B 0.000,C 90.000,E1 17.149} C_DIS
LIN {X -0.198,Y -408.445,Z 814.874,A 0.000,B 0.000,C 90.000,E1 13.355} C_DIS
END
